	AHH_Mottakstank				: BOOL;
	HH_LS_Mottakstank			: BOOL;
	AHH_Reaktor					: BOOL;
	Reaktor_2_Forrigling		: BOOL;
END_VAR
VAR_OUTPUT
	PauseOK						: BOOL;
END_VAR
VAR

END_VAR


IF Pause THEN
	IF ((AHH_Mottakstank OR HH_LS_Mottakstank ) AND NOT Reaktor_2_Forrigling AND NOT AHH_Reaktor) THEN	// forrigling mot R2
		PauseOK := TRUE;
	ELSE
		PauseOK := FALSE;
	END_IF;
END_IF;

END_FUNCTION_BLOCK

// Device/Application/fbUtrekningar
FUNCTION_BLOCK fbUtrekningar
VAR_INPUT
END_VAR
VAR_OUTPUT
END_VAR
VAR
	Reaktor1		: MA;
	Reaktor2		: MA;
END_VAR



// Sette MA innganane

// Beregne frå nivå til volum reaktor 1
VolumReaktor(Height := GVL_R1.Nivaa, Volum => GVL_R1.Volum);

// Beregne frå nivå til volum reaktor 2
VolumReaktor(Height := GVL_R1.Nivaa, Volum => GVL_R2.Volum);

END_FUNCTION_BLOCK

// Device/Application/VolumReaktor
FUNCTION VolumReaktor : REAL
VAR_INPUT
	Height			: REAL;
END_VAR

VAR_OUTPUT
	Volum			: REAL;
END_VAR

VAR CONSTANT
	Radius 			: REAL := 3.0;
	pi_value 		: REAL := 3.14;
END_VAR


Volum := Height * pi_value * Radius * Radius;

END_FUNCTION

// Device/Application/Heile_R1/Reaktor1
PROGRAM Reaktor1
VAR

	Tilstandsmaskin		: tmReaktor;

	Innpumping			: R1_Innpumping;
	Pause				: R1_Pause;
	Reaksjon			: R1_Reaksjon;
	Sedementering		: R1_Sedementering;
	Uttaping			: R1_Uttapping;
	Beregning			: fbUtrekningar;
	Slam				: R1_Slam;
END_VAR

// Tilstander for Tilstandsmaskin
Pause(TM_Pause := Tilstandsmaskin.Pause); // R1_Pause
Innpumping(TM_Innpumping := Tilstandsmaskin.Innpumping); // R1_Innpumping
Reaksjon(TM_Reaksjon := Tilstandsmaskin.Reaksjon); // R1_Reaksjon
// Tilstandsmaskin for SARA Reaktor 1
Tilstandsmaskin(
    PauseOK := Pause.TM_PauseOK,
    InnpumpingOK := Innpumping.TM_InnpumpingOK,
    ReaksjonOK := Reaksjon.TM_ReaksjonOK,
    SedementeringOK := Sedementering.TM_SedementeringOK,
    UttappingOK := Uttaping.TM_UttappingOK); // tmReaktor
GVL_R1.Pause := Tilstandsmaskin.Pause;
GVL_R1.Innpumping := Tilstandsmaskin.Innpumping;
GVL_R1.Reaksjon := Tilstandsmaskin.Reaksjon;
GVL_R1.Sedimentering := Tilstandsmaskin.Sedementering;
GVL_R1.Uttapping := Tilstandsmaskin.Uttapping;
Sedementering(TM_Sedementering := Tilstandsmaskin.Sedementering); // R1_Sedementering
Uttaping(TM_Uttapping := Tilstandsmaskin.Uttapping); // R1_Uttapping
// Slamuttak
Slam(TM_Slam := Tilstandsmaskin.Reaksjon); // R1_Slam

END_PROGRAM

// Device/Application/Heile_R1/R1_Innpumping
FUNCTION_BLOCK R1_Innpumping
VAR_INPUT
	TM_Innpumping			: BOOL;
END_VAR
VAR_OUTPUT
	TM_InnpumpingOK			: BOOL;
END_VAR

VAR
PP00_LS02   		: MB;
PP00_LS01  			: MB;
PP00_LT01	 		: MA;
PP01_LT01	 		: MA;

PP01_PS01		 	: SBE;
PP02_PS01		 	: SBE;
PP01_VP01   		: SBV;

PA01_BL01				: SBE;

Sekvens_Innpumping	: fbInnpumping;
	Sim: FBVALVESIM;
END_VAR

VAR_TEMP
	PYHR			: REAL := 100;
	PYLR			: REAL := 0;
	PP00_LT01_PAHH	: REAL := 32;
	PP00_LT01_PALL	: REAL := 5;
	PP01_LT01_PAHH	: REAL := 90;
END_VAR

// -------------------------------------------------------------------------------------------------------------------------------- INPUTS --------------------------------------------------------------------------------------------------------------------------------
// Mottakstank vippe høg
PP00_LS01(); // MB
// Mottakstank vippe lav
PP00_LS02(); // MB
// Mottakstank Nivåmåling
PP00_LT01(
    X := GVL_Inputs.PP00_LT01_X,
    PAHH := PP00_LT01_PAHH,
    PALL := PP00_LT01_PALL,
    PYHR := PYHR,
    PYLR := PYLR); // MA
// Reaktor 1 Nivåmåling
PP01_LT01(X := GVL_Inputs.PP01_LT01_X, PAHH := PP01_LT01_PAHH, PYHR := PYHR, PYLR := PYLR); // MA
// -------------------------------------------------------------------------------------------------------------------------------- CODE --------------------------------------------------------------------------------------------------------------------------------
Sekvens_Innpumping(
    Sending_Tank_AHH := PP00_LT01.AHH,
    Sending_Tank_ALL := PP00_LT01.ALL,
    Sending_Tank_LS_High := PP00_LS01.Y,
    Sending_Tank_LS_Low := PP00_LS02.Y,
    Reciving_Tank_AHH := PP01_LT01.AHH,
    Reciving_Tank_ALL := PP01_LT01.ALL,
    ValveBCH := PP01_VP01.BCH,
    ValveBCL := PP01_VP01.BCL,
    Pump1BCL := PP01_PS01.BCL,
    Pump2BCL := PP02_PS01.BCL,
    TM_Innpumping := TM_Innpumping,
    Max_Innpumpings_Tid := GVL_R1.SekvenstidInnpumping,
    Intervall_blaser_tid := GVL_R1.IntervallBlaser,
    Gangtid_Blaser := GVL_R1.GangtidBlaser); // fbInnpumping
// Reaktor 1 blåser
PA01_BL01(
    XGH := PA01_BL01.Y,
    XH := Sekvens_Innpumping.Blower_start,
    XL := Sekvens_Innpumping.Blower_stopp,
    XE := Simu.XE,
    LA := Simu.LA); // SBE
GVL_Outputs.PA01_BL01_Y := PA01_BL01.Y;
TM_InnpumpingOK := Sekvens_Innpumping.TM_InnpumpingOK;
// -------------------------------------------------------------------------------------------------------------------------------- OUTPUTS --------------------------------------------------------------------------------------------------------------------------------
// Inntaktspumpe 1
PP01_PS01(
    XGH := PP01_PS01.Y,
    XH := Sekvens_Innpumping.Pump1XH,
    XL := Sekvens_Innpumping.Pump1XL,
    XE := Simu.XE,
    LA := Simu.LA); // SBE
GVL_Outputs.PP01_PS01_Y := PP01_PS01.Y;
// Inntaktspumpe 2
PP02_PS01(
    XGH := PP02_PS01.Y,
    XH := Sekvens_Innpumping.Pump2XH,
    XL := Sekvens_Innpumping.Pump2_XL,
    XE := Simu.XE,
    LA := Simu.LA); // SBE
GVL_Outputs.PP02_PS01_Y := PP02_PS01.Y;
// Reaktor 1 inn ventil
PP01_VP01(
    XGH := Sim.BCH,
    XGL := Sim.BCL,
    XH := Sekvens_Innpumping.Valve_Open,
    XL := Sekvens_Innpumping.Valve_Close,
    LA := Simu.LA); // SBV
Sim(X := PP01_VP01.Y); // FBVALVESIM

END_FUNCTION_BLOCK

// Device/Application/Heile_R1/R1_Pause
FUNCTION_BLOCK R1_Pause
VAR_INPUT
	XE					: BOOL;			// Input from state machine
END_VAR
VAR_OUTPUT
	Y					: BOOL;			// Output to state machine
END_VAR
VAR
	// INPUT BLOCKS
	PP00_LS02   		: MB;			// Mottasktank vippe lav, call "Monitor Binary" 
	PP00_LS01  			: MB;			// Mottasktank vippe høg, call "Monitor Binary" 
	PP00_LT01	 		: MA;			// Mottasktank nivåmålar, call "Monitor Analog"
	PP01_LT01	 		: MA;			// Reaktor 1 nivåmålar,   call "Monitor Analog"

	// OUTPUT BLOCKS
	PA01_BL01			: SBE;			// Reaktor 1 blåser,	 call "Switch Binary Electrical"
	
	// FUNCTION BLOCKS
	SekvensPause		: fbPause;		// Pause logic, call "fbPause"
END_VAR
VAR_TEMP
	// FUNCTION CONTROL PARAMETERS
	PYHR				: REAL := 100;	// (Mottasktank nivåmålar & Reaktor 1 nivåmålar) MA Parameter Y high range
	PYLR				: REAL := 0;	// (Mottasktank nivåmålar & Reaktor 1 nivåmålar) MA Parameter Y low range
	PP00_LT01_PAHH		: REAL := 70;	// (Mottasktank nivåmålar) 						 MA Parameter high high action
	PP01_LT01_PAHH		: REAL := 90;	// (Reaktor 1 nivåmålar)   						 MA Parameter low low action 
END_VAR

// -------------------------------------------------------------------------------------------------------------------------------------------------IN BLOCKS----------------------------------------------------------------------------------------------------------------------------------------------------------------------------------------------------------
// Mottakstank vippe høg
// INPUTS
PP00_LS01(X := GVL_Inputs.PP00_LS01_X); // MB
// Mottakstank vippe lav
// INPUTS
PP00_LS02(X := GVL_Inputs.PP00_LS02_X); // MB
// Mottakstank Nivåmåling
// INPUTS
PP00_LT01(X := GVL_Inputs.PP00_LT01_X, PAHH := PP00_LT01_PAHH, PYHR := PYHR, PYLR := PYLR); // MA
// OUTPUTS
// OUTPUTS
// OUTPUTS
GVL_Rest.MottakstankNivaa := PP00_LT01.Y;
// Reaktor 1 Nivåmåling
// INPUTS
PP01_LT01(X := GVL_Inputs.PP01_LT01_X, PAHH := PP01_LT01_PAHH, PYHR := PYHR, PYLR := PYLR); // MA
// OUTPUTS
GVL_R1.Nivaa := PP01_LT01.Y;
// -------------------------------------------------------------------------------------------------------------------------------------------------CODE ----------------------------------------------------------------------------------------------------------------------------------------------------------------------------------------------------------
SekvensPause(
    XE := XE,
    AHH_Mottakstank := PP00_LT01.AHH,
    AHH_LS_Mottakstank := PP00_LS01.Y,
    AHH_Reaktor := PP01_LT01.AHH,
    XB := GVL_R2.Innpumping,
    PTD := GVL_R1.GangtidBlaser,
    PTI := GVL_R1.IntervallBlaser); // fbPause
// -------------------------------------------------------------------------------------------------------------------------------------------------OUT BLOCKS----------------------------------------------------------------------------------------------------------------------------------------------------------------------------------------------------------
// Reaktor 1 Blåser
// Inputs
PA01_BL01(
    XGH := PA01_BL01.Y,
    XH := SekvensPause.YH_Blower,
    XL := SekvensPause.YL_Blower,
    XE := XE,
    LA := GVL_R1.Pause); // SBE
GVL_R1.Pause_PA01_BL01 := PA01_BL01.Y;
// OUTPUTS
GVL_R1.Pause_PA01_BL01_YF := PA01_BL01.YF;
Y := SekvensPause.Y;

END_FUNCTION_BLOCK

// Device/Application/Heile_R1/R1_Reaksjon
FUNCTION_BLOCK R1_Reaksjon
VAR_INPUT
	TM_Reaksjon			: BOOL;
END_VAR
VAR_OUTPUT
	TM_ReaksjonOK			: BOOL;
END_VAR
VAR
	Reaksjon				: fbReaksjon;
	Doseringspumpe			: SBE;
	Blaser					: SBE;
END_VAR

Reaksjon(
    TM_Reaksjon := TM_Reaksjon,
    Blaser_Confirmed_stopped := Blaser.BCL,
    Max_Reaksjon_Tid := GVL_R1.SekvenstidReaksjon,
    Gangtid_Anoks := GVL_R1.GangtidAnoks,
    Gangtid_Aerob := GVL_R1.GangtidAerob,
    Gangtid_Kjemikalie := GVL_R1.GangtidKjemikalieDosering,
    DoseringStartTidForSlutt := GVL_R1.SikkerheitsIntervallKjemikalie); // fbReaksjon
TM_ReaksjonOK := Reaksjon.TM_ReaksjonOK;
Blaser(XH := Reaksjon.Start_Blaser, XL := Reaksjon.Stopp_Blaser); // SBE
Doseringspumpe(XH := Reaksjon.Start_Pumpe, XL := Reaksjon.Stopp_Pumpe); // SBE

END_FUNCTION_BLOCK

// Device/Application/Function blocks/fbReaksjon
FUNCTION_BLOCK fbReaksjon
VAR_INPUT
	TM_Reaksjon							: BOOL;			// Start frå Tilstandsmaskin
	
	Blaser_Confirmed_stopped			: BOOL;
	
	// Timer og Tider
	Max_Reaksjon_Tid					: TIME;			// Sekvenstid
	Gangtid_Anoks						: TIME;			// Gangtid uten blåsing aktiv
	Gangtid_Aerob						: TIME;			// Gangtid med blåsing aktiv
	Gangtid_Kjemikalie					: TIME;			// Gangtid for kjemikalie
	DoseringStartTidForSlutt			: TIME;
END_VAR

VAR_OUTPUT
	TM_ReaksjonOK						: BOOL;			// Til Tilstandsmaskin
	
	// Blåser
	Start_Blaser						: BOOL;
	Stopp_Blaser						: BOOL;
	
	// Kjemikalie Pumpe
	Start_Pumpe							: BOOL;
	Stopp_Pumpe							: BOOL;
END_VAR

VAR
	AnoksTimer							: fbTimer;
	AerobTimer							: fbTimer;
	ReaksjonsTimer						: fbTimer;
	KjemikalieTimer						: fbTimer;
	
	siCase	: SINT;
END_VAR

VAR CONSTANT
	ciInit	: SINT := 0;
	ciAerob : SINT := 1;
	ciAnoks : SINT := 2;
END_VAR


// INPUTS

// Timer
AnoksTimer();
AerobTimer();
ReaksjonsTimer();
KjemikalieTimer();

AnoksTimer.PTDH 		:= Gangtid_Anoks;
AerobTimer.PTDH			:= Gangtid_Aerob;
ReaksjonsTimer.PTDH 	:= Max_Reaksjon_Tid;
KjemikalieTimer.PTDH	:= Max_Reaksjon_Tid - (Gangtid_Kjemikalie + DoseringStartTidForSlutt);
KjemikalieTimer.PTDL	:= Gangtid_Kjemikalie;

// Hantering av feil større ein max tid
IF (Gangtid_Anoks > Max_Reaksjon_Tid) THEN
	Gangtid_Anoks := Max_Reaksjon_Tid;
END_IF

IF (Gangtid_Aerob > Max_Reaksjon_Tid) THEN
	Gangtid_Aerob := Max_Reaksjon_Tid;
END_IF


IF TM_Reaksjon THEN
	
	CASE siCase OF
		
		ciInit:
		
		IF NOT (TM_ReaksjonOK) THEN
			ReaksjonsTimer.X 	:= TRUE;
			KjemikalieTimer.X 	:= TRUE;
			siCase := ciAerob;
		END_IF

		ciAerob:
			
			// Reset Anoks Timer
			AnoksTimer.X := FALSE;
			
			// Start Aerob Timer
			AerobTimer.X := TRUE;
			
			// Start Blåser
			Stopp_Blaser := FALSE;
			Start_Blaser := TRUE;
			
			// Neste case
			IF (AerobTimer.Y) THEN
				siCase := ciAnoks;
			END_IF
			
		ciAnoks:
		
			// Reset Aerob Timer
			AerobTimer.X := FALSE;
			
			// Start Anoks Timer
			AnoksTimer.X := TRUE;
			
			// Stopp Blåser
			Stopp_Blaser := TRUE;
			Start_Blaser := FALSE;
			
			// Neste case
			IF (AnoksTimer.Y) THEN
				siCase := ciAerob;
			END_IF
	END_CASE

	IF (KjemikalieTimer.Y) THEN
		
		KjemikalieTimer.X := FALSE;
		
		// Kjemikalie Pumpe
		Stopp_Pumpe := FALSE;
		Start_Pumpe := TRUE;

	ELSE
		// Kjemikalie Pumpe
		Stopp_Pumpe := TRUE;
		Start_Pumpe := FALSE;
	END_IF




	IF (ReaksjonsTimer.Y) THEN
		
		// Stopp blåser og pumpe uansett tilstand
		Stopp_Blaser := TRUE;
		Start_Blaser := FALSE;
					
		IF (Blaser_Confirmed_stopped) THEN
			
			// Reset Timers
			ReaksjonsTimer.X 	:= FALSE;
			KjemikalieTimer.X 	:= FALSE;
			AnoksTimer.X		:= FALSE;
			AerobTimer.X		:= FALSE;
			
			// Send to initial state
			siCase 				:= ciInit;
			
			// Send to tilstandsmaskin
			TM_ReaksjonOK 		:= TRUE;
		END_IF
	END_IF

ELSE
	TM_ReaksjonOK := FALSE;
END_IF


// OUTPUTS

END_FUNCTION_BLOCK

// Device/Application/Heile_R1/R1_Sedementering
FUNCTION_BLOCK R1_Sedementering
VAR_INPUT
	TM_Sedementering 	: BOOL; 			// Input from state machine
END_VAR
VAR_OUTPUT
	TM_SedementeringOK 	: BOOL;				// Output to state machine
END_VAR
VAR
	// INPUT BLOCKS

	// OUTPUT BLOCKS

	// FUNCTION BLOCKS	
	Sedimentering		: fbSedementering;	// Sedimentering logic, call "fbSedimentering"
END_VAR

// -------------------------------------------------------------------------------------------------------------------------------------------------IN BLOCKS----------------------------------------------------------------------------------------------------------------------------------------------------------------------------------------------------------
// ------------------------------------------------------------------------------------------------------------------------------------------------- CODE ----------------------------------------------------------------------------------------------------------------------------------------------------------------------------------------------------------
// ------------------------------------------------------------------------------------------------------------------------------------------------- OUT BLOCKS ----------------------------------------------------------------------------------------------------------------------------------------------------------------------------------------------------------
Sedimentering(TM_Sedementering := TM_Sedementering, SedementeringTid := GVL_R1.SekvenstidSedimentering); // fbSedementering
TM_SedementeringOK := Sedimentering.TM_SedementeringOK;

END_FUNCTION_BLOCK

// Device/Application/Function blocks/fbSedementering
FUNCTION_BLOCK fbSedementering
VAR_INPUT
	XE					: BOOL;		// External enable from state machine
END_VAR
VAR_INPUT RETAIN
	PST					: TIME;		// Parameter max sedimentation time
END_VAR

VAR_OUTPUT
	Y					: BOOL;		// Function output, pulsed true when sequence is finished.
END_VAR
VAR
	SedementeringTimer		: fbTimer;
END_VAR

// ***************************************************************************************
// Copyright: Peter Søreide Skaar, Roar Bøyum, Vegard Aven Ullebø [2024]
// All rights reserved.

// This code was developed as part of a Bachelor's thesis conducted for Renasys AS 
// and Sunnfjord Kommune. 

// Unauthorized reproduction, distribution, or modification of this code, in whole 
// or in part, is strictly prohibited without the express permission of the copyright 
// holder.
// ***************************************************************************************

SedementeringTimer();
SedementeringTimer.PTDH := PST;

IF (XE) THEN
	
	SedementeringTimer.X := TRUE;
	
	IF (SedementeringTimer.Y) THEN
		
		Y := TRUE;	
	END_IF
ELSE
	Y := FALSE;	
	SedementeringTimer.X := FALSE;
END_IF

END_FUNCTION_BLOCK

// Device/Application/Heile_R1/R1_Uttapping
FUNCTION_BLOCK R1_Uttapping
VAR_INPUT
	TM_Uttapping	: BOOL;
END_VAR
VAR_OUTPUT
	TM_UttappingOK	: BOOL;
END_VAR
VAR
	Uttapping		: fbUttapping;
	TW01_VP01		: SBV;
	PP01_LT01		: MA;
	Sim: FBVALVESIM;
END_VAR
VAR_TEMP
	PYHR			: REAL := 100;
	PYLR			: REAL := 0;
	PP00_LT01_PAHH	: REAL := 32;
	PP01_LT01_PAHH	: REAL := 90;
END_VAR

PP01_LT01(X := GVL_Inputs.PP01_LT01_X, PAHH := PP01_LT01_PAHH, PYHR := PYHR, PYLR := PYLR); // MA
Simu.R1Nivaa := PP01_LT01.Y;
Uttapping(
    TM_Uttapping := TM_Uttapping,
    Max_uttaping_Tid := GVL_R1.SekvenstidUttapping,
    Tank_ALL := PP01_LT01.ALL,
    Valve_Confirmed_Close := TW01_VP01.BCL,
    Reaktor_Nivaa := PP01_LT01.Y); // fbUttapping
TM_UttappingOK := Uttapping.TM_UttappingOK;
GVL_R1.DeltaNivaaDrenert := Uttapping.DeltaNivaa;
TW01_VP01(XGH := Sim.BCH, XGL := Sim.BCL, XH := Uttapping.Valve_Open, XL := Uttapping.Valve_Close); // SBV
Simu.TW02_VH01_YF := TW01_VP01.YF;
Sim(X := TW01_VP01.Y); // FBVALVESIM
GVL_Outputs.TW01_VP01_BCH := TW01_VP01.BCH;

END_FUNCTION_BLOCK

// Device/Application/Function blocks/fbUttapping
FUNCTION_BLOCK fbUttapping
VAR_INPUT
	X						: REAL;		// Input from leveltransmitter current level reactor
	XE						: BOOL;		// External enable from state machine
	XGL						: BOOL;		// Drain valve binary confirm low	
	X1						: BOOL;		// Low level from leveltransmitter reactor
END_VAR

VAR_INPUT RETAIN
	PUT						: TIME;		// Paramter Max uttapping time
END_VAR

VAR_OUTPUT
	Y						: BOOL;		// Output to state machine, pulsed if finshed sequence
	Y1						: REAL;		// Output (DeltaLevel) StartLevel - FinishedLevel
	YHDrainValve			: BOOL;		// Output YH open drain valve
	YLDrainValve			: BOOL;		// Output YL close drain valve
END_VAR
VAR
	UttappingTimer			: fbTimer;
	sbUttap					: BOOL;
	
	PreUttapNivaa			: REAL;
	sbFlank					: BOOL;
END_VAR

VAR_TEMP
	tbFlank					: BOOL;
END_VAR

// ***************************************************************************************
// Copyright: Peter Søreide Skaar, Roar Bøyum, Vegard Aven Ullebø [2024]
// All rights reserved.

// This code was developed as part of a Bachelor's thesis conducted for Renasys AS 
// and Sunnfjord Kommune. 

// Unauthorized reproduction, distribution, or modification of this code, in whole 
// or in part, is strictly prohibited without the express permission of the copyright 
// holder.
// ***************************************************************************************

// INNPUTS

// Timers
UttappingTimer();
UttappingTimer.PTDH := PUT;

IF (XE) THEN
	
	// Start av Timer
	UttappingTimer.X := TRUE;
	
	// Only posetiv edge
	IF (XE AND NOT sbUttap) THEN
		PreUttapNivaa := X;
	END_IF

	// Open valve
	YHDrainValve 	:= TRUE;
	YLDrainValve := FALSE;

	IF (X1 OR UttappingTimer.Y) THEN
		
		// Close valve
		YLDrainValve := TRUE;
		YHDrainValve  := FALSE;
		
		IF (XGL) THEN
			
			tbFlank := TRUE;
			
			// Reset Timer
			UttappingTimer.X := FALSE;
			
			// Til Tilstandsmaskin 
			Y := TRUE;
			
			IF (tbFlank AND NOT sbFLANK) THEN
				Y1 := PreUttapNivaa - X;
			END_IF
			
			// Posetive edge retrigger;
			sbFlank := tbFlank;
			
		END_IF		
	END_IF
ELSE
	tbFlank := FALSE;
	Y := FALSE;
END_IF

// Retrigger

sbUttap := XE;

// OUTPUTS

END_FUNCTION_BLOCK

// Device/Application/Heile_R1/R1_Slam
FUNCTION_BLOCK R1_Slam
VAR_INPUT
	TM_Slam : BOOL;	
END_VAR
VAR_OUTPUT
END_VAR
VAR
	fbslamutak	: fbSlamUtak;
	PS01_VP01 	: SBV;
	PS00_VP01 	: SBV; //Sivebedventil 1
	PS00_VP02 	: SBV; //Sivebedventil 2
	PS00_VP03 	: SBV; //Sivebedventil 3
	PS00_VP04 	: SBV; //Sivebedventil 4
	
	Sim1		: fbValveSim;
	Sim2		: fbValveSim;
	Sim3		: fbValveSim;
	Sim4		: fbValveSim;
	Sim5		: fbValveSim;
END_VAR

fbSlamutak(
    X1 := GVL_R1.Nivaa,
    X2 := GVL_Rest.siSivState,
    XE := TM_Slam,
    SivValve1BCL := PS00_VP01.BCL,
    SivValve2BCL := PS00_VP02.BCL,
    SivValve3BCL := PS00_VP03.BCL,
    SivValve4BCL := PS00_VP04.BCL,
    ReactorValveBCL := PS01_VP01.BCL,
    ReactorValveBCH := PS01_VP01.BCH,
    PTI := GVL_Rest.Uttaksintervall,
    PTMT := GVL_Rest.MaxGangtidSlam,
    PRAntattSlamNivaa := GVL_Rest.AntattSlamNivaa);
GVL_Rest.PulseCoutner := fbSlamutak.Y;
// -------------------------------------------------------------------------------------------------------------------------------- OUTPUTS --------------------------------------------------------------------------------------------------------------------------------
// Reaktor Slamventil
// INPUTS
PS01_VP01(XGH := Sim1.BCH, XGL := Sim1.BCL, XH := fbSlamutak.YHReactorValve, XL := fbSlamutak.YLReactorValve); // SBV
Sim1(X := PS01_VP01.Y); // fbValveSim
// OUTPUTS
GVL_Outputs.PS01_VP01_Y := PS01_VP01.Y;
GVL_R1.PS01_VP01_YF := PS01_VP01.YF;
// Sivebed1
// INPUTS
PS00_VP01(XGH := Sim2.BCH, XGL := Sim2.BCL, XH := fbSlamutak.YHSivbed1Valve, XL := fbSlamutak.YLSivbed1Valve); // SBV
Sim2(X := PS00_VP01.Y); // fbValveSim
// OUTPUTS
GVL_R1.PS00_VP01_Y := PS00_VP01.Y;
GVL_R1.PS00_VP01_YF := PS00_VP01.YF;
// Sivebed2
// INPUTS
PS00_VP02(XGH := Sim3.BCH, XGL := Sim3.BCL, XH := fbSlamutak.YHSivbed2Valve, XL := fbSlamutak.YLSivbed2Valve); // SBV
Sim3(X := PS00_VP02.Y); // fbValveSim
// OUTPUTS
GVL_R1.PS00_VP02_Y := PS00_VP02.Y;
GVL_R1.PS00_VP02_YF := PS00_VP02.YF;
// Sivebed3
// INPUTS
PS00_VP03(XGH := Sim4.BCH, XGL := Sim4.BCL, XH := fbSlamutak.YHSivbed3Valve, XL := fbSlamutak.YLSivbed3Valve); // SBV
Sim4(X := PS00_VP03.Y); // fbValveSim
// OUTPUTS
GVL_R1.PS00_VP03_Y := PS00_VP03.Y;
GVL_R1.PS00_VP03_YF := PS00_VP03.YF;
// Sivebed4
// INPUTS
PS00_VP04(XGH := Sim4.BCH, XGL := Sim4.BCL, XH := fbSlamutak.YHSivbed4Valve, XL := fbSlamutak.YLSivbed4Valve); // SBV
Sim4(X := PS00_VP04.Y); // fbValveSim
// OUTPUTS
GVL_R1.PS00_VP04_Y := PS00_VP04.Y;
GVL_R1.PS00_VP04_YF := PS00_VP04.YF;

END_FUNCTION_BLOCK

// Device/Application/Function blocks/fbSlamutak
FUNCTION_BLOCK fbSlamutak
VAR_INPUT
	TM_Slamutak					: BOOL;	
	
	Slamalder					: INT;
	AntattSlamNivaa				: REAL;
			
	ReactorLevel				: REAL;

	SivValve1BCL				: BOOL;
	SivValve2BCL				: BOOL;
	SivValve3BCL				: BOOL;
	SivValve4BCL				: BOOL;
	
	ReactorValveBCL				: BOOL;
	ReactorValveBCH				: BOOL;
	
	Uttaksintervall				: TIME;
	MaxGangTidSlamUtak			: TIME;	
END_VAR

VAR_OUTPUT
	Y							: BOOL; //Sender pulse ferdig til sivbedHandtering for telling
	Open_Reactor_Valve			: BOOL;
	Close_Reactor_Valve			: BOOL;
	
	Open_SivCelle_1_Valve		: BOOL;
	Close_SivCelle_1_Valve		: BOOL;
	
 	Open_SivCelle_2_Valve		: BOOL;
 	Close_SivCelle_2_Valve		: BOOL;
 	
 	Open_SivCelle_3_Valve		: BOOL;
 	Close_SivCelle_3_Valve		: BOOL;
 	
 	Open_SivCelle_4_Valve		: BOOL;
 	Close_SivCelle_4_Valve		: BOOL;

END_VAR

VAR
	siSivBed					: SINT;	
	PreUttakNiva				: REAL;	
	sbUttakTimerY				: BOOL;	
	
	GangtidSlamtapping			: fbTimer;
	UttaksTimer					: fbTimer;
	SivBedTimer					: fbTimer;
	OutputPulse					: fbTimer;

	CmSlamUttak					: REAL;
	
	AktivSivCelleBCL			: BOOL;
	
END_VAR

VAR_TEMP
	tiMillis						: LINT;
	tiDays							: LINT;
END_VAR

VAR CONSTANT
	ciInit			: SINT := 0;
	ciCelle1		: SINT := 1;
	ciCelle2		: SINT := 2;
	ciCelle3		: SINT := 3;
	CiCelle4		: SINT := 4;
	PTD				: TIME := T#2S;
	
	cliMillis2Days	: LINT := 86400000;	
	
END_VAR


// Timer teller kontinuerlig om
UttaksTimer();
GangtidSlamTapping();
OutputPulse();


UttaksTimer.PTDH := Uttaksintervall;
GangtidSlamTapping.PTDH := MaxGangTidSlamUtak;
OutputPulse.PTDL := PTD;
UttaksTimer.X := TRUE;
OutputPulse.X := FALSE;

// Convert TIME to days in INT.
tiMillis := TIME_TO_INT(Uttaksintervall);
tiDays := tiMillis / cliMillis2Days;

IF (TM_Slamutak) THEN
	
	// Timer goes true and begins slamuttak
	IF (UttaksTimer.Y) THEN
		
		// Storing level of reactor tank before opening valves on posetive edge		
		IF (UttaksTimer.Y AND NOT sbUttakTimerY) THEN			
			cmSlamUttak := (tiDays * AntattSlamNivaa)/Slamalder; 	// Calculating slamuttak			
			PreUttakNiva := ReactorLevel;							// Store Reactorlevel before started sludge removal.
			GangtidSlamtapping.X := TRUE;							// Start timer 			
		END_IF		
		
		// Opne reaktor slam ventil		
		Open_Reactor_Valve := TRUE;
		Close_Reactor_Valve := FALSE;
		
		// Based on which sivcelle is in use open the respectiv valves
		// Required Reactorvalve confirmed open		
		IF (ReactorValveBCH) THEN
		
			IF (siSivBed = ciCelle1) THEN
			
				Close_Sivcelle_1_Valve 		:= FALSE;
				Open_Sivcelle_1_Valve 		:= TRUE;
			
			ELSIF (siSivBed = ciCelle2) THEN
			
				Close_Sivcelle_2_Valve 		:= FALSE;
				Open_Sivcelle_2_Valve 		:= TRUE;
			
			ELSIF (siSivBed = ciCelle3) THEN
			
				Close_Sivcelle_3_Valve 		:= FALSE;
				Open_Sivcelle_3_Valve 		:= TRUE;
		
			ELSIF (siSivBed = ciCelle4) THEN
				
				Close_Sivcelle_4_Valve 		:= FALSE;
				Open_Sivcelle_4_Valve 		:= TRUE;
			END_IF		
		END_IF
		
		// Stopping SlamUttak when the required amout of sludge is removed from the reactor
		
		IF ((ReactorLevel < (PreUttakNiva - CmSlamUttak)) OR GangTidSlamTapping.Y) THEN
			
			// Closing reactor valve
			
			Open_Reactor_Valve 		:= FALSE;
			Close_Reactor_Valve 	:= TRUE;
						
			// Closing sivcelle valves 			
			IF    (siSivBed = ciCelle1) THEN
			
				AktivSivCelleBCL := SivValve1BCL;
			
				Close_Sivcelle_1_Valve 		:= TRUE;
				Open_Sivcelle_1_Valve 		:= FALSE;
			
			ELSIF (siSivBed = ciCelle2) THEN
			
				AktivSivCelleBCL := SivValve2BCL;
			
				Close_Sivcelle_2_Valve 		:= TRUE;
				Open_Sivcelle_2_Valve 		:= FALSE;
			
			ELSIF (siSivBed = ciCelle3) THEN
			
				AktivSivCelleBCL := SivValve3BCL;
			
				Close_Sivcelle_3_Valve 		:= TRUE;
				Open_Sivcelle_3_Valve 		:= FALSE;
		
			ELSIF (siSivBed = ciCelle4) THEN
				
				AktivSivCelleBCL := SivValve4BCL;
				
				Close_Sivcelle_4_Valve 		:= TRUE;
				Open_Sivcelle_4_Valve 		:= FALSE;
			END_IF
				
				
			// If the vales are confirmed close the initial timer is reset and starts counting again		
			IF ((ReactorValveBCL AND AktivSivCelleBCL)) THEN
			
			// Resetting timer
			UttaksTimer.X 			:= FALSE;
			GangtidSlamtapping.X 	:= FALSE;			
			OutputPulse.X := TRUE;					
			END_IF		
		END_IF		
	END_IF
	
	// Posetive edge retrigger
	sbUttakTimerY := UttaksTimer.Y;	
END_IF



//Handle outputs
Y := OutputPulse.Y;

END_FUNCTION_BLOCK

// Device/Application/Heile_R2/Reaktor2
PROGRAM Reaktor2
VAR
	Tilstandsmaskin		: tmReaktor;
	Innpumping			: R1_Innpumping;
	Pause				: R1_Pause;
	Reaksjon			: R1_Reaksjon;
	Sedementering		: R1_Sedementering;
	Uttaping			: R1_Uttapping;
	Beregning			: fbCalculations;	
END_VAR

// Tilstander for Tilstandsmaskin
Pause(XE := Tilstandsmaskin.Pause); // R1_Pause
Innpumping(XE := Tilstandsmaskin.Innpumping); // R1_Innpumping
Reaksjon(XE := Tilstandsmaskin.Reaksjon); // R1_Reaksjon
// Tilstandsmaskin for SARA Reaktor 1
Tilstandsmaskin(
    PauseOK := Pause.Y,
    InnpumpingOK := Innpumping.Y,
    ReaksjonOK := Reaksjon.Y,
    SedementeringOK := Sedementering.Y,
    UttappingOK := Uttaping.Y); // tmReaktor
GVL_R1.Pause := Tilstandsmaskin.Pause;
GVL_R1.Innpumping := Tilstandsmaskin.Innpumping;
GVL_R1.Reaksjon := Tilstandsmaskin.Reaksjon;
GVL_R1.Sedimentering := Tilstandsmaskin.Sedementering;
GVL_R1.Uttapping := Tilstandsmaskin.Uttapping;
GVL_R1.State := Tilstandsmaskin.State;
Sedementering(XE := Tilstandsmaskin.Sedementering); // R1_Sedementering
Uttaping(XE := Tilstandsmaskin.Uttapping); // R1_Uttapping

END_PROGRAM

// Device/Application/Heile_R2/Reaktor2
PROGRAM Reaktor2
VAR
	Tilstandsmaskin		: tmReaktor;

	Innpumping			: R2_Innpumping;
	Pause				: R2_Pause;
END_VAR

Tilstandsmaskin(PauseOK := Pause.TM_PauseOK, InnpumpingOK := Innpumping.TM_InnpumpingOK); // tmReaktor
GVL_TM.R2_Pause := Tilstandsmaskin.Pause;
GVL_TM.R2_Innpumping := Tilstandsmaskin.Innpumping;
GVL_TM.R2_Reaksjon := Tilstandsmaskin.Reaksjon;
GVL_TM.R2_Sedementering := Tilstandsmaskin.Sedementering;
GVL_TM.R2_Uttapping := Tilstandsmaskin.Uttapping;
Innpumping(TM_Innpumping := Tilstandsmaskin.Innpumping); // R2_Innpumping
Pause(TM_Pause := Tilstandsmaskin.Pause); // R2_Pause

END_PROGRAM

// Device/Application/Heile_R2/R2_Pause
FUNCTION_BLOCK R2_Pause
VAR_INPUT
	XE					: BOOL;			// Input from state machine
END_VAR
VAR_OUTPUT
	Y					: BOOL;			// Output to state machine
END_VAR
VAR
	// INPUT BLOCKS
	PP00_LS02   		: MB;			// Mottasktank vippe lav, call "Monitor Binary" 
	PP00_LS01  			: MB;			// Mottasktank vippe høg, call "Monitor Binary" 
	PP00_LT01	 		: MA;			// Mottasktank nivåmålar, call "Monitor Analog"
	PP02_LT02	 		: MA;			// Reaktor 2 nivåmålar,   call "Monitor Analog"

	// OUTPUT BLOCKS
	PA02_BL01			: SBE;			// Reaktor 2 blåser,	 call "Switch Binary Electrical"
	
	// FUNCTION BLOCKS
	SekvensPause		: fbPause;		// Pause logic, call "fbPause"	
	PA02_BL0			: SBE;
END_VAR
VAR_TEMP
	// FUNCTION CONTROL PARAMETERS
	PYHR				: REAL := 100;	// (Mottasktank nivåmålar & Reaktor 1 nivåmålar) MA Parameter Y high range
	PYLR				: REAL := 0;	// (Mottasktank nivåmålar & Reaktor 1 nivåmålar) MA Parameter Y low range
	PP00_LT01_PAHH		: REAL := 32;	// (Mottasktank nivåmålar) 						 MA Parameter high high action
	PP02_LT02_PAHH		: REAL := 90;	// (Reaktor 2 nivåmålar)   						 MA Parameter low low action 
END_VAR

// -------------------------------------------------------------------------------------------------------------------------------------------------IN BLOCKS----------------------------------------------------------------------------------------------------------------------------------------------------------------------------------------------------------
// Mottakstank vippe høg
// INPUTS
PP00_LS01(X := GVL_Inputs.PP00_LS01_X); // MB
// Mottakstank vippe lav
// INPUTS
PP00_LS02(X := GVL_Inputs.PP00_LS02_X); // MB
// Mottakstank Nivåmåling
// INPUTS
PP00_LT01(X := GVL_Inputs.PP00_LT01_X, PAHH := PP00_LT01_PAHH, PYHR := PYHR, PYLR := PYLR); // MA
// OUTPUTS
// OUTPUTS
// OUTPUTS
GVL_Rest.MottakstankNivaa := PP00_LT01.Y;
// Reaktor 2 Nivåmåling
// INPUTS
PP02_LT02(X := GVL_Inputs.PP02_LT02_X, PAHH := PP02_LT02_PAHH, PYHR := PYHR, PYLR := PYLR); // MA
// OUTPUTS
GVL_R2.Nivaa := PP02_LT02.Y;
// -------------------------------------------------------------------------------------------------------------------------------------------------CODE ----------------------------------------------------------------------------------------------------------------------------------------------------------------------------------------------------------
SekvensPause(
    XE := XE,
    AHH_Mottakstank := PP00_LT01.AHH,
    AHH_LS_Mottakstank := PP00_LS01.Y,
    AHH_Reaktor := PP02_LT02.AHH,
    XB := GVL_R1.Innpumping,
    PTD := GVL_R2.GangtidBlaser,
    PTI := GVL_R2.IntervallBlaser); // fbPause
// -------------------------------------------------------------------------------------------------------------------------------------------------OUT BLOCKS----------------------------------------------------------------------------------------------------------------------------------------------------------------------------------------------------------
// Reaktor 2 Blåser
// Inputs
PA02_BL01(
    XGH := PA02_BL01.Y,
    XH := SekvensPause.YH_Blower,
    XL := SekvensPause.YL_Blower,
    XE := XE,
    LA := GVL_R2.Pause); // SBE
GVL_R2.Pause_PA01_BL01 := PA02_BL01.Y;
// OUTPUTS
GVL_R2.Pause_PA01_BL01_YF := PA02_BL01.YF;
Y := SekvensPause.Y;

END_FUNCTION_BLOCK

// Device/Application/Heile_R2/R2_Pause
FUNCTION_BLOCK R2_Pause
VAR_INPUT
	TM_Pause			: BOOL;
END_VAR
VAR_OUTPUT
	TM_PauseOK			: BOOL;
END_VAR
VAR
	PP00_LS01	: MB;
	PP00_LS02	: MB;
	PP00_LT01	: MA;
	PP01_LT01	: MA;
	
	SekvensPause	: fbPause;	
END_VAR

PP00_LS01(); // MB
PP00_LS02(); // MB
PP00_LT01(); // MA
PP01_LT01(); // MA
SekvensPause(
    Pause := TM_Pause,
    AHH_Mottakstank := PP00_LT01.AHH,
    HH_LS_Mottakstank := PP00_LS01.Y,
    AHH_Reaktor := PP01_LT01.AHH,
    Reaktor_2_Forrigling := GVL_TM.R1_Innpumping); // fbPause
TM_PauseOK := SekvensPause.PauseOK;

END_FUNCTION_BLOCK

// Device/Application/Heile_R2/R2_Innpumping
FUNCTION_BLOCK R2_Innpumping
VAR_INPUT
	TM_Innpumping			: BOOL;
END_VAR
VAR_OUTPUT
	TM_InnpumpingOK			: BOOL;
END_VAR

VAR
PP00_LS02   		: MB;
PP00_LS01  			: MB;
PP00_LT01	 		: MA;
PP01_LT01	 		: MA;

PP01_PS01		 	: SBE;
PP02_PS01		 	: SBE;
PP01_VP01   		: SBV;

Sekvens_Innpumping	: fbInnpumping;

END_VAR

PP00_LS01(); // MB
PP00_LS02(); // MB
PP00_LT01(); // MA
PP01_LT01(); // MA
Sekvens_Innpumping(
    Sending_Tank_AHH := PP00_LT01.AHH,
    Sending_Tank_ALL := PP00_LT01.ALL,
    Sending_Tank_LS_High := PP00_LS01.Y,
    Sending_Tank_LS_Low := PP00_LS02.Y,
    Reciving_Tank_AHH := PP01_LT01.AHH,
    Reciving_Tank_ALL := PP01_LT01.ALL,
    ValveBCH := PP01_VP01.BCH,
    ValveBCL := PP01_VP01.BCL,
    Pump1BCL := PP01_PS01.BCL,
    Pump2BCL := PP02_PS01.BCL,
    TM_Innpumping := TM_Innpumping); // fbInnpumping
TM_InnpumpingOK := Sekvens_Innpumping.TM_InnpumpingOK;
PP01_VP01(XH := Sekvens_Innpumping.Valve_Open, XL := Sekvens_Innpumping.Valve_Close); // SBV
PP01_PS01(XH := Sekvens_Innpumping.Pump1XH, XL := Sekvens_Innpumping.Pump1XL); // SBE
PP02_PS01(XH := Sekvens_Innpumping.Pump2XH, XL := Sekvens_Innpumping.Pump2_XL); // SBE

END_FUNCTION_BLOCK

// Device/Application/Heile_R2/R2_Innpumping
FUNCTION_BLOCK R2_Innpumping
VAR_INPUT
	XE						: BOOL;			// Input from state machine
END_VAR
VAR_OUTPUT
	Y						: BOOL;			// Output to state machine
END_VAR

VAR
	// INPUT BLOCKS
	PP00_LS02   			: MB;			// Mottasktank vippe lav, call "Monitor Binary" 
	PP00_LS01  				: MB;			// Mottasktank vippe høg, call "Monitor Binary" 
	PP00_LT01	 			: MA;			// Mottasktank nivåmålar, call "Monitor Analog"
	PP01_LT01	 			: MA;			// Reaktor 2 nivåmålar,   call "Monitor Analog"
	
	// OUTPUT BLOCKS
	PA01_BL01				: SBE;			// Reaktor 2 blåser,	 call "Switch Binary Electrical"
	PP01_PS01		 		: SBE;			// Matepumpe 1,			 call "Switch Binary Electrical"
	PP02_PS01		 		: SBE;			// Matepumpe 2,			 call "Switch Binary Electrical"
	PP01_VP01   			: SBV;			// Reaktor 2 inn ventil, call "Switch Binary Valve"
	
	// FUNCTION BLOCKS
	Sekvens_Innpumping		: fbInnpumping;	// Innpumping logic,         call "fbInnpumping"
	Sim						: fbValveSim;	// Feedback balve simulator, call "fbValveSim"
	PA02_BL01				: SBE;
	PP02_VP01				: SBV;
	PP02_LT02				: MA;

END_VAR

VAR_TEMP		
	// FUNCTION CONTROL PARAMETERS
	PYHR					: REAL := 100;		// (Mottasktank nivåmålar & Reaktor 2 nivåmålar) MA Parameter Y high range
	PYLR					: REAL := 0;		// (Mottasktank nivåmålar & Reaktor 2 nivåmålar) MA Parameter Y low range
	PP00_LT01_PBXH			: REAL := 70;		// (Mottasktank nivåmålar) 						 MA Parameter high high action
	PP00_LT01_PBXL			: REAL := 10;		// (Mottasktank nivåmålar) 						 MA Parameter low low action
	PP02_LT02_PBXH			: REAL := 90;		// (Reaktor 2 nivåmålar)   						 MA Parameter high high action
	END_VAR

// -------------------------------------------------------------------------------------------------------------------------------------------------IN BLOCKS----------------------------------------------------------------------------------------------------------------------------------------------------------------------------------------------------------
// Mottakstank vippe høg
// INPUTS
// OUTPUTS
PP00_LS01(X := GVL_Inputs.PP00_LS01_X); // MB
// Mottakstank vippe lav
// INPUTS
PP00_LS02(X := GVL_Inputs.PP00_LS02_X); // MB
// Mottakstank Nivåmåling
// INPUTS
PP00_LT01(
    X := GVL_Inputs.PP00_LT01_X,
    PBXH := PP00_LT01_PBXH,
    PBXL := PP00_LT01_PBXL,
    PYHR := PYHR,
    PYLR := PYLR); // MA
// OUTPUTS
// OUTPUTS
GVL_Rest.MottakstankNivaa := PP00_LT01.Y;
// Reaktor 2 Nivåmåling
// INPUTS
PP02_LT02(X := GVL_Inputs.PP02_LT02_X, PBXH := PP02_LT02_PBXH, PYHR := PYHR, PYLR := PYLR); // MA
// OUTPUTS
GVL_R2.Nivaa := PP02_LT02.Y;
// ------------------------------------------------------------------------------------------------------------------------------------------------- CODE ----------------------------------------------------------------------------------------------------------------------------------------------------------------------------------------------------------
Sekvens_Innpumping(
    X1_SendingTank := PP00_LT01.BXH,
    X2_SendingTank := PP00_LT01.BXL,
    X3_SendingTank := PP00_LS01.Y,
    X4_Sending_Tank := PP00_LS02.Y,
    X5_ReceivingTank := PP02_LT02.BXH,
    X6_ReceivingTank := PP02_LT02.BXL,
    X7_RValve := PP02_VP01.BCH,
    X8_RValve := PP02_VP01.BCL,
    X9_Pump1 := PP01_PS01.BCL,
    X10_Pump2 := PP02_PS01.BCL,
    XE := XE,
    PIT := GVL_R2.SekvenstidInnpumping,
    PTI := GVL_R2.IntervallBlaser,
    PTD := GVL_R2.GangtidBlaser); // fbInnpumping
// Reaktor 2 blåser
// INPUTS
PA02_BL01(
    XGH := PA02_BL01.Y,
    XH := Sekvens_Innpumping.YH_Blower,
    XL := Sekvens_Innpumping.YL_Blower,
    XE := GVL_R2.Innpumping,
    LA := Simu.LA); // SBE
GVL_R2.Innpumping_PA01_BL01_YF := PA02_BL01.YF;
Y := Sekvens_Innpumping.Y;
// ------------------------------------------------------------------------------------------------------------------------------------------------- OUT BLOCKS  ----------------------------------------------------------------------------------------------------------------------------------------------------------------------------------------------------------
// Inntaktspumpe 1
// INPUTS
PP01_PS01(
    XGH := PP01_PS01.Y,
    XH := Sekvens_Innpumping.YH_Pump1,
    XL := Sekvens_Innpumping.YL_Pump1,
    XE := GVL_R2.Innpumping,
    LA := Simu.LA); // SBE
GVL_R2.PP01_PS01_YF := PP01_PS01.YF;
// OUTPUTS
GVL_R2.PP01_PS01_Y := PP01_PS01.Y;
// Inntaktspumpe 2
// INPUTS
PP02_PS01(
    XGH := PP02_PS01.Y,
    XH := Sekvens_Innpumping.YH_Pump2,
    XL := Sekvens_Innpumping.YL_Pump2,
    XE := GVL_R2.Innpumping,
    LA := Simu.LA); // SBE
// OUTPUTS
GVL_R2.PP02_PS01_Y := PP02_PS01.Y;
GVL_R2.PP02_PS01_YF := PP02_PS01.YF;
// OUTPUTS
GVL_R2.Innpumping_PA02_BL01 := PA02_BL01.Y;
// Reaktor 2 inn ventil
// INPUTS
PP02_VP01(
    XGH := Sim.BCH,
    XGL := Sim.BCL,
    XH := Sekvens_Innpumping.YH_RValve,
    XL := Sekvens_Innpumping.YL_RValve,
    LA := Simu.LA); // SBV
// OUTPUTS
GVL_Outputs.PP02_VP01_Y := PP02_VP01.Y;
GVL_R2.PP01_VP01_YF := PP02_VP01.YF;
GVL_R2.PP01_VP01_BCH := PP02_VP01.BCH;
Sim(X := PP02_VP01.Y); // FBVALVESIM

END_FUNCTION_BLOCK

// Device/Application/Heile_R2/R2_Reaksjon
FUNCTION_BLOCK R2_Reaksjon
VAR_INPUT
	XE					: BOOL;			// Input from state machine
END_VAR
VAR_OUTPUT
	Y					: BOOL; 		// Output to state machine
END_VAR
VAR
	// INPUT BLOCKS

	// OUTPUT BLOCKS
	CH00_PH01			: SBE;			// Reaktor 2 doseringspumpe, call "Switch Binary Electrical"
	PA01_BL01			: SBE;			// Reaktor 2 blåser,	 	 call "Switch Binary Electrical"
	Slam				: R1_Slam;		// Slammuttak
	
	// FUNCTION BLOCKS
	Reaksjon			: fbReaksjon;	// Reaksjon logic, call "fbReaksjon"
	PA02_BL01			: SBE;			// Blower R2
	CH00_PH02			: SBE;			// ChemPump R2
END_VAR

// note: 2 stored wires end on pins the file does not list and are not shown
// Slamuttak
Slam(XE := XE); // R1_Slam
// -------------------------------------------------------------------------------------------------------------------------------------------------IN BLOCKS----------------------------------------------------------------------------------------------------------------------------------------------------------------------------------------------------------
// ------------------------------------------------------------------------------------------------------------------------------------------------- CODE ----------------------------------------------------------------------------------------------------------------------------------------------------------------------------------------------------------
Reaksjon(
    XE := XE,
    XHLBlower := PA02_BL01.BCL,
    PRT := GVL_R2.SekvenstidReaksjon,
    PTAN := GVL_R2.GangtidAnoks,
    PTAE := GVL_R2.GangtidAerob,
    PTCP := GVL_R2.GangtidKjemikalieDosering,
    PTCR := GVL_R2.SikkerheitsIntervallKjemikalie); // fbReaksjon
Y := Reaksjon.Y;
// ------------------------------------------------------------------------------------------------------------------------------------------------- OUT BLOCKS ----------------------------------------------------------------------------------------------------------------------------------------------------------------------------------------------------------
// Reaktor 2 Blåser
// INPUTS
PA02_BL01(XH := Reaksjon.YHBlower, XL := Reaksjon.YLBlower, XE := GVL_R2.Reaksjon, LA := Simu.LA); // SBE
GVL_R2.Reaksjon_PA01_BL01_YF := PA02_BL01.YF;
// OUTPUTS
GVL_R2.Reaksjon_PA01_BL01 := PA02_BL01.Y;
// Reaktor 2 Doseringspumpe
// INPUTS
CH00_PH02(
    XGH := CH00_PH02.Y,
    XH := Reaksjon.YHChemPump,
    XL := Reaksjon.YLChemPump,
    XE := GVL_R2.Reaksjon,
    LA := Simu.LA); // SBE
GVL_R2.CH00_PH02_YF := CH00_PH02.YF;
// OUTPUTS
GVL_Outputs.CH00_PH02_Y := CH00_PH02.Y;

END_FUNCTION_BLOCK

// Device/Application/Heile_R2/R2_Sedementering
FUNCTION_BLOCK R2_Sedementering
VAR_INPUT
	XE 					: BOOL; 			// Input from state machine
END_VAR
VAR_OUTPUT
	Y 					: BOOL;				// Output to state machine
END_VAR
VAR
	// INPUT BLOCKS

	// OUTPUT BLOCKS

	// FUNCTION BLOCKS	
	Sedimentering		: fbSedementering;	// Sedimentering logic, call "fbSedimentering"
END_VAR

// -------------------------------------------------------------------------------------------------------------------------------------------------IN BLOCKS----------------------------------------------------------------------------------------------------------------------------------------------------------------------------------------------------------
// ------------------------------------------------------------------------------------------------------------------------------------------------- CODE ----------------------------------------------------------------------------------------------------------------------------------------------------------------------------------------------------------
// ------------------------------------------------------------------------------------------------------------------------------------------------- OUT BLOCKS ----------------------------------------------------------------------------------------------------------------------------------------------------------------------------------------------------------
Sedimentering(XE := XE, PST := GVL_R2.SekvenstidSedimentering); // fbSedementering
Y := Sedimentering.Y;

END_FUNCTION_BLOCK

// Device/Application/Heile_R2/R2_Uttapping
FUNCTION_BLOCK R2_Uttapping
VAR_INPUT
	XE	: BOOL;				 // Input from state machine
END_VAR
VAR_OUTPUT
	Y				: BOOL; // Output to state machine
END_VAR
VAR
	// INPUT BLOCKS
	PP01_LT01		: MA; 	// Reaktor 1 nivåmålar,   call "Monitor Analog"
	
	// OUTPUT BLOCKS
	TW01_VP01		: SBV;	// Reaktor 1 dreneringsventil, call "Switch Binary Valve"
	
	// FUNCTION BLOCKS
	Uttapping		: fbUttapping;
	Sim				: FBVALVESIM;
	PP02_LT02		: MA;
	TW02_VP01		: SBV;
	PP02_LT022_PALL: INT;
END_VAR
VAR_TEMP
	PYHR			: REAL := 100;
	PYLR			: REAL := 0;	
	PP02_LT02_PAHH	: REAL := 90;
	PP02_LT02_PALL	: REAL := 90;
	
END_VAR

// ------------------------------------------------------------------------------------------------------------------------------------------------- IN BLOCKS ----------------------------------------------------------------------------------------------------------------------------------------------------------------------------------------------------------
// Reaktor 2 Nivåmålar
// INPUTS
PP02_LT02(
    X := GVL_Inputs.PP02_LT02_X,
    PAHH := PP02_LT02_PAHH,
    PALL := PP02_LT022_PALL,
    PYHR := PYHR,
    PYLR := PYLR); // MA
// OUTPUTS
GVL_R2.Nivaa := PP02_LT02.Y;
// ------------------------------------------------------------------------------------------------------------------------------------------------- CODE  ----------------------------------------------------------------------------------------------------------------------------------------------------------------------------------------------------------
Uttapping(
    XE := XE,
    PUT := GVL_R2.SekvenstidUttapping,
    ALL := PP02_LT02.ALL,
    XGL := TW02_VP01.BCL,
    X := PP02_LT02.Y); // fbUttapping
Y := Uttapping.Y;
GVL_R2.DeltaNivaaDrenert := Uttapping.Y1;
// ------------------------------------------------------------------------------------------------------------------------------------------------- OUTPUT BLOCKS ----------------------------------------------------------------------------------------------------------------------------------------------------------------------------------------------------------
// Reaktor 2 dreneringsventil
// INPUTS
TW02_VP01(
    XGH := Sim.BCH,
    XGL := Sim.BCL,
    XH := Uttapping.YHDrainValve,
    XL := Uttapping.YLDrainValve,
    LA := Simu.LA); // SBV
GVL_R2.TW01_VH01_YF := TW02_VP01.YF;
Sim(X := TW02_VP01.Y); // FBVALVESIM
// OUTPUTS
GVL_Outputs.TW02_VP01_Y := TW02_VP01.Y;

END_FUNCTION_BLOCK

// Device/Application/IEC_Time
FUNCTION IEC_Time : BOOL
VAR_INPUT
	Start : BOOL;
END_VAR

VAR
END_VAR

END_FUNCTION

// Device/Application/POU
PROGRAM POU
VAR
	test : BOOL;
	test2 : BOOL;
END_VAR

END_PROGRAM

// Device/Application/SBV_ReArranged
FUNCTION_BLOCK SBV_ReArranged
VAR_INPUT
	XGH            : BOOL;                		 // eXternal Feedback Position High
    XGL            : BOOL;                		 // eXternal Feedback Position Low
    XH             : BOOL;                		 // eXternal Switch to Position High - in automatic mode
    XL             : BOOL;                		 // eXternal Switch to Position Low - in automatic mode
	XOH            : BOOL;               		 // eXternal Switch to Posistion High - in local/outside mode
	XOL            : BOOL;               		 // eXternal Switch to Posistion Low - in local/outside mode
	XF             : BOOL;                 		 // eXternal Fault 
	LSH            : BOOL;               		 // Lock Safeguard High
	LSL            : BOOL;               		 // Lock Safeguard Low
	FSH            : BOOL;                		 // Force Safeguarding High
    FSL            : BOOL;                		 // [Priority] Force Safeguarding Low
    FDH            : BOOL;              		 // Force Disable High
    FDL            : BOOL;             		     // [Priority] Force Disable Low
	FB             : BOOL;             		     // Force Block	
	FU             : BOOL;						 // Force Supression
	LA             : BOOL;               		 // Set Auto
	LM             : BOOL;               		 // [Priority 2]Set Manual
	LO             : BOOL;               		 // [Priority 1]Set Outside
    //RX             : BOOL;               		 // Reset Fault	
END_VAR

VAR_INPUT RETAIN 								// 
    PFFD           	: TIME := T#5S;       		// Feedback failure delay
    PTDH           	: TIME := T#5S;        	  	// Transit delay low to high
    PTDL           	: TIME := T#5S;       		// Transit delay high to low
    PSTO           	: BOOL;               		// Output YH and YL  constant on.
	PTTO			: TIME := T#2000MS;			// PULS output open YH
	PTTC			: TIME := T#2000MS;			// PULS output close YL
	PAOF			: INT  := 0;				// Parameter action on fault.
	PFT				: INT  := 3;				// Parameter feedback type
	PSUS			: INT  := 0;				// Parameter Template Startup State 
	PSUM			: INT  := 0;				// Parameter for mode at startup
	PSLO			: INT  := 0;				// Parameter for setting local or outside mode
END_VAR

VAR_OUTPUT
	Y              : BOOL;                		// 
	YH             : BOOL;               		// Normal output to switch control element to high state
    YL             : BOOL;                		// Normal output to switch control element to low state
    YF             : BOOL;                		// Control element fault
    BCH            : BOOL;               		// Binary status confirmed high
    BCL            : BOOL;                		// Binary status confirmed low
	BS             : BOOL;                		// Binary status safeguarding
	BB             : BOOL;                		// Binary status blocked
	BU             : BOOL;               		// Binary status suppressed
    BA             : BOOL;               		// Binary status automatic mode
	BO             : BOOL;                		// 
   // BM             : Bool := true;        	// Binary status manual mode    
   // BD             : Bool;                	// Binary status disabled
    YFI            : INT;               		// Fault information
END_VAR

VAR RETAIN
	
	sbBA           		 : BOOL;               	// Binary status automatic mode, RETAINED for prevstate.

END_VAR


VAR
	siState       		 : INT;                 // State of controlled element
    siNextState   		 : INT;                 // Next state of controlled element
	
	sbLA				: BOOL;					// Set auto variable
	sbLM				: BOOL;					// Set manual variable
	
	OS_FB				: BOOL;					// HMI Force block
	OS_FU				: BOOL;					// HMI Force supress
	OS_XLM				: BOOL;					// HMI Set low
	OS_XHM				: BOOL;					// HMI Set high
	
	TimerTransLow		: fbTimer;				// Timer trans low error
	TimerTransHigh		: fbTimer;				// Timer trans high erreor
	TimerFeedbackLow	: fbTimer;				// Timer no feedback low error
	TimerFeedbackHigh	: fbTimer;				// Timer no feedback high error
	OutputPulsHigh		: TP;
	OutputPulsLow		: TP;
	
	
	sbYF            : BOOL;						// Output fault variable
	sbBUpos			: BOOL;						// Binary supressed posetive flank variable
	sbBUneg			: BOOL;						// Binary supressed negative flank variable
	
	siFBlastvalue	: INT;						// 
END_VAR

VAR_TEMP

	tbHighCommand  		: BOOL;                 // High command
    tbLowCommand   		: BOOL;                 // Low Command
	tbOutsideLocal		: BOOL;					// Interlock of starting object when in local mode
	
	// INPUTS
	tbXGH            : BOOL;                	// eXternal Feedback Position High variable
    tbXGL            : BOOL;                	// eXternal Feedback Position Low variable
    tbXH             : BOOL;                	// eXternal Switch to Position High - in automatic mode variable
    tbXL             : BOOL;                	// eXternal Switch to Position Low - in automatic mode variable
	tbXOH            : BOOL;               		// eXternal Switch to Position High - In outside mode variable
	tbXOL            : BOOL;               		// eXternal Switch to Position LOW - In outside mode variable
	tbXF             : BOOL;                 	// eXternal Fault variable
	tbLSH            : BOOL;               		// Lock Safeguard High variable 
	tbLSL            : BOOL;               		// Lock Sagefuard Low variable 
	tbFSH            : BOOL;                	// Force Safeguarding High
    tbFSL            : BOOL;                	// [Priority] Force Safeguarding Low
    tbFDH            : BOOL;              		// Force Disable High
    tbFDL            : BOOL;             		// [Priority] Force Disable Low
	tbFB             : BOOL;             		// Force Blocking variable
	tbFU             : BOOL;					// Force Supression variable
	tbLA             : BOOL;               		// Lock Auto variable
	tbLM             : BOOL;               		// Lock Manuell variable
	tbLO             : BOOL;               		// Lock Outside
	
	
	// OUTPUTS
	tbY             : BOOL;                		// Output
	tbYH            : BOOL;               		// Normal output to switch control element to high state
    tbYL            : BOOL;                		// Normal output to switch control element to low state    
    tbBCH           : BOOL;               		// Binary status confirmed high
    tbBCL           : BOOL;                		// Binary status confirmed low
	tbBS            : BOOL;                		// Binary status safeguarding
	tbBB            : BOOL;                		// Binary status blocked
	tbBU            : BOOL;               		// Binary status supressed
	tbBO            : BOOL;                		// Binary status outside
	tiYFI			: INT;						// FAULT REGISTER
	
END_VAR

VAR CONSTANT
	ciInitState         : INT := 0;             // [FSM] Initial State of Control Element
    ciLow               : Int := 1;             // [FSM] Control Element in Low state
    ciTransitHigh       : Int := 2;             // [FSM] Control Element in transit to High state
    ciHigh              : Int := 3;             // [FSM] Control Element in High state
    ciTransitLow        : INT := 4;             // [FSM] Control Element in transit to Low state
	
	ciNoFault           : INT := 0;                  // [FAULT] No Fault Indication
    ciFeedbackFaultHigh : Int := 1;             // [FAULT] Feedback Fault
    ciFeedbackFaultLow  : Int := 2;             // [FAULT] Feedback Fault
    ciTransitHighFault  : Int := 3;             // [FAULT] Transit High Fault
    ciTransitLowFault   : INT := 4;             // [FAULT] Transit Low Fault
	ciExternalFault		: INT := 5;				// [FAULT] External fault
	ciConflictFault		: INT := 6;				// [FAULT] Conflict fault (Safeguard and blocking)
	ciSafeguardFault	: INT := 7;				// [FAULT] [Priority] Safeguard fault (No feedback while executing safeguard command)
	
	ciNoAction			: INT := 0;				// [PAOF] Parameter action on fault - No action
	ciClose				: INT := 1;				// [PAOF] Parameter action on fault - Closed action
	ciOpen				: INT := 2;				// [PAOF] Parameter action on fault - Open action
	
	ciNoFeedback		: INT := 0;				// [PFT] Parameter feedback mode - No feedback
	ciHighFeedback		: INT := 1;				// [PFT] Parameter feedback mode - High feedback
	ciLowFeedback		: INT := 2;				// [PFT] Parameter feedback mode - Low feedback
	ciFullFeedback		: INT := 3;				// [PFT] Parameter feedback mode - Full feedback
	
	ciStartupClosed		: INT := 0;				//
	ciStartupOpen		: INT := 1;
	ciStartupFeedback	: INT := 2;
	
	ciModeStartupManual		: INT := 0;			// Sets the mode of the block at startup
	ciModeStartupAuto		: INT := 1;			// Sets the mode of the block at startup
	ciModeStartupPrev		: INT := 2;			// Sets the mode of the block at startup
	
	ciModeLocal				: INT := 0;			// Parameter for setting local mode
	ciModeOutside			: INT := 1;			// Parameter for setting outside mode
END_VAR

//INFO, COPYRIGHT MANGOIPA GROUP INC
//SBV function block


//Populate Temporaries and preset outputs

tbXGH 									:= XGH;
tbXGL 									:= XGL;    
tbXH									:= XH;            
tbXL									:= XL;   
tbXOH									:= XOH;     
tbXOL									:= XOL;           
tbXF									:= XF;            
tbLSH									:= LSH;           
tbLSL									:= LSL;           
tbFSH									:= FSH;           
tbFSL									:= FSL;            
tbFDH									:= FDH;            
tbFDL									:= FDL;            
tbFB									:= FB;            
tbFU									:= FU;            
tbLA									:= LA;              
tbLM									:= LM;             
tbLO									:= LO;       

// Timers
TimerTransLow();													// Timer for transition to low fault
TimerTransHigh();													// Timer for transition to high fault
TimerFeedbackLow();													// Timer for no feedback low fault
TimerFeedbackHigh();												// Timer for no feedback high fault
OutputPulsHigh();										 			// Timer for puls YH
OutputPulsLow();													// Timer for puls YL

//Timer parameters (should be behind a restart/startup function))
TimerTransLow.PTDH						:= PTDH;
TimerTransHigh.PTDH 					:= PTDL;
TimerFeedbackLow.PTDH					:= PFFD;
TimerFeedbackHigh.PTDH					:= PFFD;
OutputPulsHigh.PT						:= PTTO;
OutputPulsLow.PT						:= PTTC;


// Handle external faults, subject to supression
IF (tbXF AND NOT tbFU) THEN
	tiYFI 								:= ciExternalFault;
END_IF

// Handle High output puls YH / YL
IF NOT (siState = ciTransitHigh) THEN
	OutputPulsHigh.IN 					:= FALSE;
END_IF

IF NOT (siState = ciTransitLow) THEN
	OutputPulsLow.IN 					:= FALSE;
END_IF


// MODECONTROLL
// Mode Control - AUTO/MAN
IF tbLM AND NOT sbLM  THEN
    sbBA                       			:= FALSE;					// Manual mode, BA = 0
ELSIF tbLA AND NOT sbLA THEN
    sbBA                       			:= TRUE; 	    			// Auto mode posetive edge,	BA = 1
END_IF;
	
sbLA 									:= tbLA;					// Retrigger posetive edge for Mode Control.
sbLM 									:= tbLM;					// Retrigger posetive edge for Mode Control.

// Mode Controll - Outside/Local mode.
IF tbLO THEN		
	tbBO 								:= TRUE;					// Sets status outside and force off auto-mode
	sbBA 								:= FALSE;	
	
	CASE PSLO OF													// Case for Parameter for setting local/outside
	ciModeLocal:	
		tbOutsideLocal				    := TRUE;					// Switches the block between High and Low in local mode from XGH/XGL
		IF tbXGH THEN	
			siState 					:= ciHigh;
		ELSIF tbXGL THEN			
			siState					    := ciLow;
		END_IF
				
	ciModeOutside: 													// If in outside mode, XOH/XOL will controll the block
	tbOutsideLocal 						:= FALSE;
	//
	END_CASE
ELSE
	tbBO 								:= FALSE;							
END_IF	

// SAFEGUARDING (Stod tidligere over modecontroll.)
// Handle lock safeguard mode, subject to blocking
IF (tbLSL AND NOT tbFB) THEN
	sbBA 								:= FALSE;					// Set mode to manual
ELSIF (tbLSH AND NOT tbFB) THEN
	sbBA 								:= FALSE;					// Set mode to manual
END_IF

// Handling safeguarding BS status, triggered by any Safeguarding
IF (tbLSH OR tbLSL OR tbFSH OR tbFSL) THEN
	tbBS 								:= TRUE;
ELSE
	tbBS 								:= FALSE;
END_IF

// Handling blocking BB status
IF (tbFB OR OS_FB) THEN
	tbBB 								:= TRUE;
ELSE
	tbBB 								:= FALSE;
END_IF

//Blocking blocks safeguard and disable transition modes
IF tbBB THEN
	tbLSL 								:= FALSE;
	tbLSH							    := FALSE;
	tbFSL 								:= FALSE;
	tbFSH 								:= FALSE;
	tbFDH 								:= FALSE;
	tbFDL 								:= FALSE;
END_IF

// Handle conlfict fault when safeguarding and blocking. ( Stod tidligre under low & high command)
IF (tbBS AND tbBB) THEN
	tiYFI 							    := ciConflictFault;
END_IF

// SUPRESSION
// Handling supression BU status ON/OFF
IF (tbFU OR OS_FU) THEN
	tbBU  								:= TRUE;	
ELSE
	tbBU 								:= FALSE;
END_IF

// Handles supression and PFT (Parameter feedback type)
IF tbBU AND NOT sbBUpos THEN
	siFBlastvalue 						:= PFT;						// Stores PFT before supression sets to "no feedback" on posetive edge
	PFT									:= ciNoFeedback;
END_IF

IF NOT tbBU AND sbBUneg THEN										// sets PFT to last value on negative edge
	PFT 								:= siFBlastValue;
END_IF

sbBUpos									:= tbBU;					// Posetive edge retrigger
sbBUneg 								:= tbBU;    				// Negative edge retrigger

//LOW AND HIGH COMMAND
//High and low commands evaluation (AUTO & MANUAL & OUTSIDE & LSL & LSH FDL & FDH
tbLowCommand                 		    := (tbXL AND sbBA) OR 										// Auto 
								 		   (OS_XLM AND NOT sbBA AND NOT tbBO) OR 					// Manuell (Triggered by XLM supressed by Auto & Outside mode)
								 		   (tbBO AND tbXOL AND NOT tbOutsideLocal) OR 				// Outside (Triggered by XOL if in not local outside mode)	
								 		   (tbLSL AND NOT tbFB) OR									// Lock Safeguard Low subject by blocking
								 		   (tbFSL AND NOT tbFB);									// Force safeguard Low subject by blocking
												

tbHighCommand                 			:= (tbXH AND sbBA) OR 										// Auto
								           (OS_XHM AND NOT sbBA AND NOT tbBO AND NOT tbBS) OR 		// Manuell (Triggered by XLM supressed by Auto & Outside mode
								           (tbBO AND tbXOH AND NOT tbOutsideLocal) OR 				// Outside (Triggered by XOL if in not local outside mode)
								           (tbLSH AND NOT tbFB) OR									// Lock Safeguard Low subject by blocking
								           (tbFSH AND NOT tbFB);									// Force safeguard Low subject by blocking
											

										   
// Handle force disable high command and low command
IF tbFDH AND NOT tbFB THEN
    tbHighCommand            			:= FALSE;   				//If FDH is true then erase high command, prevent transit to high
END_IF;

IF tbFDL AND NOT tbFB THEN
    tbLowCommand             			:= FALSE;   				//If FDL is true then erase low command, prevent transit to low
END_IF;

// Handle Force safeguard commands
IF tbFSL THEN
    tbHighCommand            			:= FALSE;
    tbLowCommand              			:= NOT tbXGL;    			// As long as FSL is true and not correct feedback, force transit to low
	
ELSIF tbFSH THEN													// I manuell skal den ha Y = 0 (lukka) etter FSL er ute. (Høgkant OS_XLH?)
    tbHighCommand             			:= NOT tbXGH;   			// As long as FSH is true and not correct feedback, force transit to high
    tbLowCommand              			:= FALSE;	
// I manuell skal den ha Y = 1 (lukka) etter FSL er ute.
END_IF;


// Handle parameter action on fault
IF sbYF THEN
	CASE PAOF OF 
		ciNoAction:									   			     // No action on fault			
			sbYF 						:= sbYF;		
		ciClose:													 // Close
			tbLowCommand 				:= TRUE;		
		ciOpen:														 // Open
			tbHighCommand 				:= TRUE;		
	END_CASE	
END_IF


// Handle parameter feedbacks - Sets the mode of feedback
CASE PFT OF
	ciNoFeedback:
		tbXGH 							:= (siState = ciHigh) OR (siState = ciTransitHigh);	// If no feedback mode, the state sets the XGH/XGL direct			
		tbXGL 							:= (siState = ciLOW)  OR (siState = ciTransitlow);
	ciHighFeedback:
		tbXGL 							:= (siState = ciLOW)  OR (siState = ciTransitlow);	// If no High feedback, the transition or low state sets XGL direct
	ciLowFeedback:
		tbXGH 							:= (siState = ciHigh) OR (siState = ciTransitHigh);	// If no High feedback, the transition or high state sets XGH direct
	ciFullFeedback:
		tbXGH 							:= tbXGH;
		tbXGL := tbXGL;
END_CASE;


//Determine next state
IF tbHighCommand THEN
    siNextState              		    := ciHigh;
ELSIF tbLowCommand THEN
    siNextState              		    := ciLow;
End_If;


//Tilstandsmaskina 
CASE siState OF 
	//INIT STATE
	ciInitState:														// Initial state, sets some parameters for startup
	
	CASE PSUM OF														// Sets the Statup mode.
			ciModeStartupManual		: 
				sbBA 					:= FALSE;
							
			ciModeStartupAuto		: 
				sbBA 					:= TRUE;	
		
			ciModeStartupPrev		: 
				sbBA 					:= sbBA;
	END_CASE
	
	//Sets the startup state of the block - Parameter Template Startup State
	CASE PSUS OF														
		ciStartupClosed		:  
			siState := ciLow;
			
		ciStartupOpen		:  
			siState := ciHigh;
			
		ciStartupFeedback	:  											// If feedback state, XGL/XGH determines the start state of the block
			IF tbXGH THEN
				siState					:= ciHigh;
			ELSIF XGL THEN
				siState 				:= ciLow;		
			END_IF
	END_CASE
	
	// Case for handling next state
	CASE siNextState OF
		ciHigh: 
			siState						:= ciTransitHigh;
			
		ciLow :	
			siState 		 			:= ciTransitLow;		
	END_CASE	
	
	// LOW STATE 
	ciLow:	
	
		IF (NOT tbXGL OR tbXGH) THEN									// Faulthandling if no feedback detected	
		    TimerFeedbackLow.X := TRUE;
	
            IF TimerFeedbackLow.Y THEN									// Starts the timer if missing feedback detected
                tiYFI           		:= ciFeedbackFaultLow;
            END_IF;
        ELSE
            TimerFeedbackLow.X := FALSE;								// Resets timer if feedback returns
        End_If;

        CASE siNextState OF												// Sets the next state
            ciHigh :                
                siState      		 	:= ciTransitHigh;
        END_CASE;
	
	// TRANSIT HIGH STATE	
	ciTransitHigh:
		
		TimerTransHigh.X 				:= TRUE;						// Sets timer for allowed time before feedback
		OutputPulsHigh.IN 			    := TRUE;						// Sets timer for puls output
				
		IF tbXGH THEN													// Feedback detected, resets timers and changes state
			TimerTransHigh.X 		    := FALSE;
			siState           		    := ciHigh;
		END_IF			
	
		IF (TimerTransHigh.Y) THEN										// Handles no feedback fault
			tiYFI						:= ciTransitHighFault;
		END_IF
		
		CASE siNextState OF												// Changes state 
            ciLow :                
                siState     		    := ciTransitLow;
        End_Case;
		
	ciHigh:
	//HIGH STATE	
	    IF (NOT tbXGH OR tbXGL) THEN									// Faulthandling when no feedback			
            TimerFeedbackHigh.X 		:= TRUE;						// Starts timer when no feedback
			
            IF TimerFeedbackHigh.Y THEN									// Faulthandling of timer
                tiYFI           		:= ciFeedbackFaultHigh;
            END_IF;
        ELSE
            TimerFeedbackHigh.X 		:= FALSE;						// Resets timer if feedback returns
        End_If;
		
        CASE siNextState OF												// Changes states 
            ciLow :
                siState       		  	:= ciTransitLow;
        End_Case;
	
	ciTransitLow:
	//TRANSIT LOW STATE
		TimerTransLow.X 				:= TRUE;						// Starts timer for transit 
		OutputPulsLow.IN 				:= TRUE;						// Starts timer for pulse YL
	
		IF tbXGL THEN	
			TimerTransLow.X 			:= FALSE;						// Reset timer if feedback
			siState          			:= ciLOW;						// Changes from transit to Low 
		END_IF
		
			IF (TimerTransLow.Y) THEN									// Faulthandling if no feedback
				tiYFI					:= ciTransitLowFault;	
			END_IF
		
		CASE siNextState OF												// Changes states 
            ciHigh :                
                siState      		 	:= ciTransitHigh;
        End_Case;	

END_CASE

// Safeguard fault if safeguard and no feedback fault
IF (tbBS AND ((tiYFI = ciFeedbackFaultHigh) OR (tiYFI = ciFeedbackFaultLow))) THEN
	tiYFI 							    := ciSafeguardFault;
END_IF;

// FAULT handling
sbYF 									:= (tiYFI > ciNoFault);

//Handle supression of YF
IF tbBU THEN
	sbYF							    := FALSE;
END_IF


//Write to output //TATT FRA OLAV DIREKTE
Y										:= 	(siState = ciTransitHigh) OR ((siState = ciHigh));
YH                            			:=	OutputPulsHigh.Q OR (PSTO AND (siState = ciTransitHigh)) ;
YL                           			:= 	OutputPulsLow.Q OR (PSTO AND (siState = ciTransitLow)) ;
BA										:= 	sbBA;
BU										:=  tbBU;
YF                           			:= 	(sbYF);
YFI										:=  tiYFI;
BCH                          			:= 	(siState = ciHigh) AND tbXGH AND NOT tbXGL;
BCL                         			:= 	(siState = ciLow) AND tbXGL AND NOT tbXGH;
BS										:=  tbBS;

//Write to HMI

END_FUNCTION_BLOCK

// Device/Application/test_SFC
PROGRAM test_SFC
VAR
END_VAR

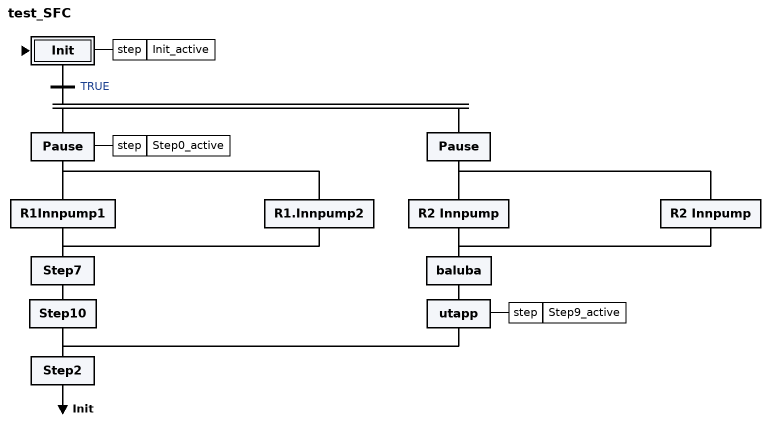
INITIAL_STEP Init:
    Init_active(N);  // step action
END_STEP
TRANSITION FROM Init TO (Pause, Pause)
    := TRUE;
END_TRANSITION
STEP Pause:
    Step0_active(N);  // step action
END_STEP
// no transition between Pause and R1Innpump1
// no transition between Pause and R1.Innpump2
STEP R1Innpump1:
END_STEP
// no transition between R1Innpump1 and Step7
STEP R1_Innpump2:  // name as stored: R1.Innpump2
END_STEP
// no transition between R1.Innpump2 and Step7
STEP Step7:
END_STEP
// no transition between Step7 and Step10
STEP Step10:
END_STEP
// no transition between Step10 and Step2
STEP Pause:
END_STEP
// no transition between Pause and R2 Innpump
// no transition between Pause and R2 Innpump
STEP R2_Innpump:  // name as stored: R2 Innpump
END_STEP
// no transition between R2 Innpump and baluba
STEP R2_Innpump:  // name as stored: R2 Innpump
END_STEP
// no transition between R2 Innpump and baluba
STEP baluba:
END_STEP
// no transition between baluba and utapp
STEP utapp:
    Step9_active(N);  // step action
END_STEP
// no transition between utapp and Step2
STEP Step2:
END_STEP
// no transition between Step2 and Init
// branch label varInnpumpOK
// branch label VarInnpumpok2

ACTION Init_active:

END_ACTION

END_PROGRAM

// Device/Application/tmReactor1
FUNCTION_BLOCK tmReactor1
VAR_INPUT
//  	PP00_LT01_AHH				: BOOL;					// Mottaktstank nivåmåler
//  	PP00_LT01_ALL				: BOOL;					// Mottaktstank nivåmåler
//  	PP00_LS02					: BOOL;					// Inngang for vippe i mottakstank HIGH HIGH
//  	PP00_LS01					: BOOL;					// Inngang for vippe i mottakstank LOW LOW 		
//  	PP01_LT01					: BOOL;					// Reaktor 1 nivå¨måler
END_VAR

VAR_OUTPUT	

END_VAR

VAR_TEMP	
	//Innputs
	tbXE							: BOOL;
	tblt_Mottakstank_AHH			: BOOL;						// ER Høg om nivå er over tillatt innpumping
	tblt_Mottakstank_ALL			: BOOL;						// ER Høg om nivå er over tillatt innpumping
	tbls_hog						: BOOL;
	tbls_lav						: BOOL;	

	//Output
	tbPause						: BOOL;							//
	tbInnpumping 				: BOOL;
	tbInnpumping_Pause			: BOOL;
	tbReaksjon 					: BOOL;
	tbSedementering 			: BOOL;
	tbUttapping					: BOOL;
	
END_VAR


VAR
	siState						: INT;		
	sitest 						: INT;
	InnpumpingTimer				: fbTimer;
	ReaksjonTimer				: fbTimer;
	SedimenteringTimer			: fbTimer;
	UttappingTimer				: fbTimer;
	
	Pause						: fbPause;
	Innpumping					: fbInnpumping;
END_VAR


VAR CONSTANT
	ciInit				     	: INT := 0;		
	ciPause			     		: INT := 1;						
	ciInnpumping 		     	: INT := 2;		
	ciInnpumping_Pause			: INT := 3;		
	ciReaksjon 			     	: INT := 4;		
	ciSedementering 		    : INT := 5;		
	ciUttapping			 	    : INT := 6;	
		
END_VAR

//Tilstandsmaskin som styrer 1 reaktor.

 //tblt_Mottakstank_AHH			:= PP00_LT01_AHH;
 //tblt_Mottakstank_ALL			:= PP00_LT01_ALL;
 //tbls_hog						:= PP00_LS02;
 //tbls_lav						:= PP00_LS01;

//Timer
InnpumpingTimer();
ReaksjonTimer();
SedimenteringTimer();	
UttappingTimer();

//Setter tid til timere - Må endres til GVB på ett tidspunkt.
InnpumpingTimer.PTDH				:= GVL_Sekvenstider.TidInnpumpingMaks;
ReaksjonTimer.PTDH 					:= GVL_Sekvenstider.TidReaksjon;
SedimenteringTimer.PTDH				:= GVL_Sekvenstider.TidSedimentering;	
UttappingTimer.PTDH					:= GVL_Sekvenstider.TidUttapping;


CASE siState OF
	ciInit:
		//Setter timere 
		siState 					:= ciPause;
		
	ciPause	:	
		tbPause 					:= TRUE;
		
		//Reset av timers	
		InnpumpingTimer.X				:= FALSE;
		ReaksjonTimer.X					:= FALSE;
		SedimenteringTimer.X			:= FALSE;	
		UttappingTimer.X				:= FALSE;	
		
		//Pause();
		
		IF GVL_TM.PauseReaktor1OK THEN	// forrigling mot R2
			siState 				:= ciInnpumping;
		END_IF	
	
	 
	ciInnpumping :	
	//	
		tbInnpumping 						:= TRUE;		
		
		//Innpumping();
				
		IF (GVL_TM.InnpumpingReaktor1OK) THEN
			siState 						:= ciReaksjon;
		END_IF
				
		
// 		InnpumpingTimer.X					:= TRUE;
// 		IF (PP01_LT01 OR InnpumpingTimer.Y ) THEN									// Eller timer
// 			siState 						:= ciReaksjon;
// 		END_IF
// 		
// 		IF (PP00_LT01_ALL OR PP00_LS01) THEN
// 			siState := ciInnpumping_Pause;
// 		END_IF
	
// 	ciInnpumping_Pause: 	
// 	//	
// 		tbInnpumping_Pause 					:= TRUE;
// 		IF (tblt_Mottakstank_AHH OR tbls_hog ) THEN								
// 			siState 						:= ciInnpumping;
// 		END_IF
// 		
// 		IF InnpumpingTimer.Y THEN
// 			siState 						:= 	ciReaksjon;
// 		END_IF
		
	ciReaksjon: 	
	//	
		tbReaksjon 							:= TRUE;
		ReaksjonTimer.X						:= TRUE;
		
		IF (ReaksjonTimer.Y) THEN
			siState 						:= ciSedementering;
		END_IF
		
	ciSedementering : 	
	//	
		tbSedementering 					:= TRUE;
		SedimenteringTimer.X				:= TRUE;
		
		IF (SedimenteringTimer.Y) THEN
			siState 						:= ciUttapping;
		END_IF
		
	ciUttapping	: 			
	//	
		tbUttapping 						:= TRUE;
		UttappingTimer.X					:= TRUE;
		
		IF (UttappingTimer.Y) THEN
			siState 						:= ciPause;
		END_IF

END_CASE




//Outputs
GVL_TM.Pause1						:= tbPause;
GVL_TM.Innpumping1 					:= tbInnpumping;
GVL_TM.Innpumping_Pause1		 		:= tbInnpumping_Pause;
GVL_TM.Reaksjon1 					:= tbReaksjon;
GVL_TM.Sedementering1 				:= tbSedementering;
GVL_TM.Uttapping1					:= tbUttapping;

END_FUNCTION_BLOCK

// Device/Application/Utrekningar
PROGRAM Utrekningar
VAR
	sjekk	: 			REAL;
END_VAR


// Beregne frå nivå til volum reaktor 1
VolumReaktor(Height := GVL_R1.Nivaa, Volum => GVL_R1.Volum);


// Beregne frå nivå til volum reaktor 2
VolumReaktor(Height := GVL_R1.Nivaa, Volum => GVL_R1.Volum);

END_PROGRAM

// Device/Application/Common_Functions/CommonFunctions
PROGRAM CommonFunctions
VAR
	Utrekning 				: fbCalculations;
	SivbedRotation 		    : fbSivbedRotation;
	Databehandling			: fbDataprocessing;
	O_Map					: Output_Mapping;
	HoyB					: fbHighload;
	ProcessedWater					: fbProcessedWater;
END_VAR

Utrekning(); // fbCalculations
SivbedRotation(
    X := GVL_Rest.PulseCoutner,
    X2 := GVL_Rest.GangerPrSivBed,
    XE1 := GVL_Rest.ActiveCelle1,
    XE2 := GVL_Rest.ActiveCelle2,
    XE3 := GVL_Rest.ActiveCelle3,
    XE4 := GVL_Rest.ActiveCelle4); // fbSivbedRotation
GVL_Rest.siSivState := SivbedRotation.Y;
// Bool input frå GVL
Databehandling(
    X0 := GVL_Outputs.PP01_PS01_Y,
    X1 := GVL_Outputs.PP02_PS01_Y,
    X2 := GVL_Outputs.PA01_BL01_Y,
    X3 := GVL_Outputs.PA02_BL01_Y,
    X4 := GVL_Outputs.CH00_PH01_Y,
    X5 := GVL_Outputs.CH00_PH02_Y,
    X6 := GVL_Outputs.RET_PHUS_Y,
    X7 := GVL_Outputs.DRE_PHUS_Y); // fbDatabehandling
GVL_Rest.PP02_PS01_Tottid := Databehandling.Y1;
GVL_Rest.PA01_BL01_Tottid := Databehandling.Y2;
GVL_Rest.PA02_BL01_Tottid := Databehandling.Y3;
GVL_Rest.CH00_PH01_Tottid := Databehandling.Y4;
GVL_Rest.CH00_PH02_Tottid := Databehandling.Y5;
GVL_Rest.RET_PHUS_Tottid := Databehandling.Y6;
GVL_Rest.DRE_PHUS_Tottid := Databehandling.Y7;
// Tider output til GVL
GVL_Rest.PP01_PS01_Tottid := Databehandling.Y0;
O_MAP(); // OUTPUT_MAPPING
HoyB(X := GVL_REST.MottakstankNivaa, PXR := GVL_REST.LimitHoybelastning); // fbHighload
GVL_Rest.HoyBelastning := HoyB.Y;
GVL_Rest.AntattTilrenning := HoyB.YG;
ProcessedWater(X1 := GVL_R1.DeltaKubikkDrenert, X2 := GVL_R2.DeltaKubikkDrenert); // fbProcessedWater
GVL_Rest.TotaltBehandlaVatn := ProcessedWater.Y1;
GVL_Rest.TotYear := ProcessedWater.Y2;
GVL_Rest.TotMonth := ProcessedWater.Y3;
GVL_Rest.TotWeek := ProcessedWater.Y4;
GVL_Rest.TotDay := ProcessedWater.Y5;
GVL_Rest.LastYear := ProcessedWater.Y6;
GVL_Rest.LastMonth := ProcessedWater.Y7;
GVL_Rest.LastWeek := ProcessedWater.Y8;
GVL_Rest.LastDay := ProcessedWater.Y9;

END_PROGRAM

// Device/Application/Function blocks/fbSivbedRotation
FUNCTION_BLOCK fbSivbedRotation
VAR_INPUT
	X					: BOOL;		// Normal functuon input, pulsed each time a reactor goes throigh slamtapping sequence
	XE1					: BOOL;		// Enable for rotation sivbed 1
	XE2					: BOOL;		// Enable for rotation sivbed 2
	XE3					: BOOL;		// Enable for rotation sivbed 3
	XE4					: BOOL;		// Enable for rotation sivbed 4
END_VAR

VAR_INPUT RETAIN
	X2					: INT;		// Input interger value that decides how many slamcycels one sivbed has before it rotates
END_VAR

VAR_OUTPUT
	Y					: SINT;		// Output integer value that outputs wich sivbed is currently in rotation
END_VAR

VAR
	SiSivBed			: SINT;
	siTeller			: INT;
	sbPulseCounter		: BOOL;
END_VAR

VAR CONSTANT
	ciInit				: SINT := 0;
	ciCelle1			: SINT := 1;
	ciCelle2			: SINT := 2;
	ciCelle3			: SINT := 3;
	CiCelle4			: SINT := 4;
END_VAR

//Handles the rotation of Sivebed, based on amount sivebed is used, counted from Reaktors



//Handle count of sivbed 
IF (X AND NOT sbPulseCounter) THEN	
	siTeller := siTeller + 1;			// Increase count by 1;
END_IF

sbPulseCounter := X;


IF (siTeller > X2) THEN
	siSivBed := siSivBed + 1;
	siTeller := 0;
END_IF


CASE (SiSivBed) OF
			
			ciInit:	
			
				SiSivBed := ciCelle1;
			
			ciCelle1:			
			// Sender vidare dersom Sivbed er tatt ut av drift				
				IF NOT (XE1) THEN
					SiSivBed := ciCelle2;
				END_IF
						
			ciCelle2:			
			// Sender vidare dersom Sivbed er tatt ut av drift	
				IF NOT (XE2) THEN
					SiSivBed := ciCelle3;
				END_IF
			
			ciCelle3:		
			// Sender vidare dersom Sivbed er tatt ut av drift	
				IF NOT (XE3) THEN
					SiSivBed := ciCelle4;
				END_IF
			
			ciCelle4:		
			// Sender vidare dersom Sivbed er tatt ut av drift		
				IF NOT (XE4) THEN
					SiSivBed := ciCelle1;
				END_IF
		
ELSE
	SiSivBed := ciCelle1;		
END_CASE

// OUTPUT
Y			:= siSivbed;

END_FUNCTION_BLOCK

// Device/Application/Function blocks/fbDatabehandling
FUNCTION_BLOCK fbDatabehandling
VAR_INPUT
	X0	: BOOL;
	X1	: BOOL;
	X2	: BOOL;
	X3	: BOOL;
	X4	: BOOL;
	X5	: BOOL;
	X6	: BOOL;
	X7	: BOOL;

END_VAR
VAR_OUTPUT

	Y0 : TIME;	
	Y1 : TIME;	
	Y2 : TIME;	
	Y3 : TIME;	
	Y4 : TIME;	
	Y5 : TIME;	
	Y6 : TIME;
	Y7 : TIME;	
	
END_VAR
VAR
	PP01_PS01		: fbCAC;	// Innpumpe nr 1
	PP02_PS01		: fbCAC;	// Innpumpe nr 2
	PA01_BL01		: fbCAC;	// Blåser 1
	PA02_BL01		: fbCAC;	// Blåser 2
	CH00_PH01		: fbCAC;	// Doseringspumpe 1
	CH00_PH02		: fbCAC;	// Doseringspumpe 2
	RET_PHUS		: fbCAC;	// Return på Pumpehus og sivbed
	DRE_PHUS		: fbCAC;	// Til resepient Pumpehus
END_VAR

// Time teller for innpumpe Nr 1
PP01_PS01();
PP01_PS01.X := X0;
Y0 := PP01_PS01.Tid;

// Time teller for innpumpe Nr 1
PP02_PS01();
PP02_PS01.X := X1;
 Y1 := PP02_PS01.Tid;

// Time teller for blåser 1
PA01_BL01();
PA01_BL01.X := X2;
Y2 := PA01_BL01.Tid;

// Time teller for blåser 2
PA02_BL01();
PA02_BL01.X := X3;
Y3 := PA02_BL01.Tid;

// Time teller for doseringspumpe 1
CH00_PH01();
CH00_PH01.X	:= X4;
Y4 := CH00_PH01.Tid;

// Time teller for doseringspumpe 2
CH00_PH02();
CH00_PH02.X	:= X5;
Y5 := CH00_PH02.Tid;

// Time teller for return på sivbed
RET_PHUS();
RET_PHUS.X := X6;
Y6 := RET_PHUS.Tid;

// Time teller for drenering mot resepient på sivbed
DRE_PHUS();
DRE_PHUS.X := X7;
Y7 := DRE_PHUS.Tid;

END_FUNCTION_BLOCK

// Device/Application/Function blocks/fbCAC
FUNCTION_BLOCK fbCAC
VAR_INPUT
	X			: BOOL;
END_VAR
VAR_OUTPUT
	Y  				: BOOL;			// Limit violation	

	Tid			: TIME;
	Dager		: INT;
	Timer		: INT;
	Minutt		: INT;
	Sekund		: INT;
	
	TotTimer	: LINT;
END_VAR
VAR
	stTimeOn 		: TIME;
	stTimeOff 		: TIME;
	sbDelayBlock    : BOOL;			//Beskyttelse
	sbY				: BOOL;
	sbX				: BOOL;
	
	Gangtid			: TIME;
END_VAR
VAR RETAIN
	TotalTid		: TIME;
END_VAR

VAR_TEMP
	
	// TEMP INPUTS
	tbX				: BOOL;	
	
	ttNow 			: TIME;
	ttTimeOn 		: TIME;
	ttTimeOff 		: TIME;
	
	tiMillis		: LINT;
	
	tiSekund		: LINT;
	tiMinutt		: LINT;
	tiTimer			: LINT;
	tiDays			: LINT;
	tiTotTimer		: LINT;
	tiRestMillis	: LINT;
	

END_VAR

VAR CONSTANT
	cliMillis2Days : LINT := 86400000;
	cliMillis2Hours : LINT := 3600000;
	cliMillis2Minutes : LINT := 60000;
	cliMillis2Seconds : LINT := 1000;

END_VAR

// ***************************************************************************************
// Copyright: Peter Søreide Skaar, Roar Bøyum, Vegard Aven Ullebø [2024]
// All rights reserved.

// This code was developed as part of a Bachelor's thesis conducted for Renasys AS 
// and Sunnfjord Kommune. 

// Unauthorized reproduction, distribution, or modification of this code, in whole 
// or in part, is strictly prohibited without the express permission of the copyright 
// holder.
// ***************************************************************************************


// INPUTS
tbX 								:= X;

// ttNow gets PLC time
ttNow 								:= TIME();							

// ttTime teller tida
ttTimeON 							:= ttNow - stTimeOn;
ttTimeOff 							:= ttNow - stTimeOff;

// OnDelay
IF tbX THEN
	sbDelayBlock 					:= FALSE;

	sbY 							:= TRUE;
	Gangtid := (ttTimeON-ttTimeOFF);	

ELSE	
	sbDelayBlock 					:= TRUE;
	stTimeOn  						:= ttNow;
END_IF;

// OffDelay
IF NOT tbX AND sbDelayBlock THEN
	
	sbY 							:= FALSE;
					
ELSE
	stTimeOff  							:= ttNow;	
END_IF;

// Negativ flanke på X, køyrest ein gong og tid lagrast til totaltida.

IF NOT tbX AND sbX THEN
	TotalTid := TotalTid + Gangtid;
	
	// Conversion of time from TIME variable to DAYS / HOURS / MINUTES / SECONDS
	
	tiMillis 		:= TIME_TO_LINT(TotalTid);
	
	tiDays 			:= tiMillis / cliMillis2Days;
	tiRestMillis 	:= tiMillis - (tiDays * CliMillis2Days);
	
	tiTotTimer		:= tiMillis / cliMillis2Hours;
	
	tiTimer := tiRestMillis / cliMillis2Hours;
	tiRestMillis 	:= tiRestMillis - (tiTimer * CliMillis2Hours);
	
	tiMinutt := tiRestMillis / cliMillis2Minutes;
	tiRestMillis 	:= tiRestMillis - (tiMinutt * CliMillis2Minutes);
	
	tiSekund := tiRestMillis / cliMillis2Seconds;
	tiRestMillis 	:= tiRestMillis - (tiSekund * CliMillis2Seconds);
	
END_IF

// Negativ flank retrigger
sbX := tbX;


// OUTPUTS
Y 										:= sbY;
Tid										:= TotalTid;
Dager									:= LINT_TO_INT(tiDays);
Timer									:= LINT_TO_INT(tiTimer);
Minutt									:= LINT_TO_INT(tiMinutt);
Sekund									:= LINT_TO_INT(tiSekund);
TotTimer								:= tiTotTimer;

END_FUNCTION_BLOCK

// Device/Application/Function blocks/Output_Mapping
FUNCTION_BLOCK Output_Mapping
VAR_INPUT
END_VAR
VAR_OUTPUT
END_VAR
VAR
END_VAR


// Handle all blower PA01_BL01 run signal to one output
GVL_Outputs.PA01_BL01_Y := GVL_R1.Pause_PA01_BL01 OR GVL_R1.Innpumping_PA01_BL01 OR GVL_R1.Reaksjon_PA01_BL01;

// Handle all blower PA02_BL01 run signal to one output


// Handle all matepumpe 1 run signals to one output
GVL_Outputs.PP01_PS01_Y := GVL_R1.PP01_PS01_Y OR GVL_R2.PP01_PS01_Y;

// Handle all matepumpe 2 run signals to one output
GVL_Outputs.PP02_PS01_Y := GVL_R1.PP02_PS01_Y OR GVL_R2.PP02_PS01_Y;

// Handle all sivcelle 1 valve open to one output
GVL_Outputs.PS00_VP01_Y := GVL_R1.PS00_VP01_Y OR GVL_R2.PS00_VP01_Y;

// Handle all sivcelle 2 valve open to one output
GVL_Outputs.PS00_VP02_Y := GVL_R1.PS00_VP02_Y OR GVL_R2.PS00_VP02_Y;

// Handle all sivcelle 3 valve open to one output
GVL_Outputs.PS00_VP03_Y := GVL_R1.PS00_VP03_Y OR GVL_R2.PS00_VP03_Y;

// Handle all sivcelle 4 valve open to one output
GVL_Outputs.PS00_VP04_Y := GVL_R1.PS00_VP04_Y OR GVL_R2.PS00_VP04_Y;

END_FUNCTION_BLOCK

// Device/Application/Function blocks/fbHighload
FUNCTION_BLOCK fbHighload
VAR_INPUT
	X						: REAL;

END_VAR

VAR_INPUT RETAIN
	PXR						: REAL;
END_VAR


VAR_OUTPUT
	Y						: BOOL;
	YG						: REAL;
END_VAR
VAR
	Timer					: fbTimer;
	sbY						: BOOL;
	srSample				: REAL;
	srLastSample			: REAL;
	srDelta					: REAL;
	trDelta					: REAL;
	
	FIFO					: ARRAY[1..ciArraySize] OF REAL;
	
	teller					: INT;
//END_VAR

//VAR_TEMP
	Sum						: REAL;
	Avarage					: REAL;
END_VAR

VAR CONSTANT
	SampleTime				: TIME		:= T#1M;
	crMottakstankBreidde	: REAL		:= 6.0;
	crMottakstankLengde		: REAL		:= 6.0;
	ciArraySize				: INT		:= 30;
END_VAR

//Measure over 30mins and calculates the avrage flow over 60mins


// Initialize timer
Timer();
Timer.PTDH 					:= SampleTime;

// Start timer
Timer.X 					:= TRUE;

// Saves sampled value each time timer goes true
IF (Timer.Y AND NOT sbY) THEN

	// Resetting sum
	SUM := 0;

	// Reads current value
	srSample				:= X;		
	srDelta					:= srSample - srLastSample;	
	trDelta 				:= srDelta * crMottakstankBreidde * crMottakstankLengde;
	
	// Protection against "Innpumping" negative trend.
	IF (trDelta < 0) THEN
		trDelta 			:= 0;
	END_IF
	
	
	// Moves all values in array 1 next	
	FOR teller := (ciArraySize - 1) TO 1 BY -1 DO
		FIFO[teller + 1]	:= FIFO[teller];
	END_FOR
	
	//Add into array
	FIFO[1] 				:= trDelta;
	
	// Store value
	srLastSample 			:= srSample;
	
	
	// Calculate the avarage delta across the FIFO 30min	
	FOR teller := 1 TO ciArraySize DO
		SUM 				:= SUM + FIFO[Teller];
	END_FOR	
	
	Avarage 				:= SUM / ciArraySize;
	
	// Calculates flow/hour
	YG 		:= Avarage *2;
	
	IF (YG > PXR) THEN
		Y 		:= TRUE;
	ELSE
		Y 		:= FALSE;
	END_IF
	
	IF (Y) THEN		
		// Endre sekvenstider		
		GVL_R1.SekvenstidReaksjon 		:= GVL_R1.SekvenstidReaksjonHoyg;
		GVL_R1.SekvenstidSedimentering 	:= GVL_R1.SekvenstidSedimenteringHoyg;
	ELSE
		// Vanlege sekvenstider		
		GVL_R1.SekvenstidReaksjon 		:= GVL_R1.SekvenstidReaksjonLav;
		GVL_R1.SekvenstidSedimentering 	:= GVL_R1.SekvenstidSedimenteringLav;				
	END_IF
	
	// Reset timer
	Timer.X 				:= FALSE;
END_IF


//Reset posetiv edge detection
sbY							:= Timer.Y;

END_FUNCTION_BLOCK

// Device/Application/Common_Functions/Pumphouse
FUNCTION_BLOCK Pumphouse
VAR_INPUT
END_VAR
VAR_OUTPUT
END_VAR
VAR
	//Fjernet logikblokk for pumpehus pga feilsøking.
	DrenPump	: SBE;
	ReturPump	: SBE;	
	Vippe_1		: MB;
	Vippe_2 	: MB; 
	Vippe_3		: MB;
END_VAR

Vippe_3(); // MB
Vippe_1(); // MB
Vippe_2(); // MB
DrenPump(); // SBE
Drenpump(); // SBE

END_FUNCTION_BLOCK

// Device/Application/Function blocks/Fault_Mapping
FUNCTION_BLOCK Fault_Mapping
VAR_INPUT
END_VAR
VAR_OUTPUT
END_VAR
VAR
END_VAR

END_FUNCTION_BLOCK

// Device/Application/Function blocks/fbBehandlaVatn
FUNCTION_BLOCK fbBehandlaVatn
VAR_INPUT
END_VAR
VAR_OUTPUT
END_VAR
VAR
END_VAR

END_FUNCTION_BLOCK

// Device/Application/Function blocks/fbFeilhandtering
FUNCTION_BLOCK fbFeilhandtering
VAR_INPUT
END_VAR
VAR_OUTPUT
END_VAR
VAR
END_VAR


// Collecting all faults to one fault output
// Here logic should be added what do when faults accur

END_FUNCTION_BLOCK

// Device/Application/Function blocks/fbPumphouse
FUNCTION_BLOCK fbPumphouse
VAR_INPUT
END_VAR
VAR_OUTPUT
END_VAR
VAR
END_VAR

END_FUNCTION_BLOCK

// Device/Application/Function blocks/fbPumpInterlock
FUNCTION_BLOCK fbPumpInterlock
VAR_INPUT
	X1					: BOOL;			// eXternal input1
	X2					: BOOL;			// eXternal input2
	XF					: BOOL;			// eXternal fault
END_VAR
VAR_OUTPUT
	Y1					: BOOL;			// Output
	Y2					: BOOL;			// Output
	YF					: BOOL;			// Output Fault
END_VAR

VAR
	Timer1				: fbTimer;		// Timer to hold the output
	Timer2				: fbTimer;		// Timer to hold the output
	sbX1				: BOOL;			// Static memory eXternal 
	sbX2				: BOOL;			// Static memory eXternal 
	siSwapCase		    : SINT;			// Static int Case
END_VAR

VAR_TEMP
	tbX1				: BOOL;			// temp eXternal input1
	tbX2				: BOOL;			// temp eXternal input2
	tbXF				: BOOL;			// eXternal fault			
	tbY1				: BOOL;			// temp output
	tbY2				: BOOL;			// temp output
END_VAR

VAR CONSTANT
	ciOutput1			: SINT := 1;		// constant case output 1
	ciOutput2			: SINT := 2;		// constant case output 2
	ciTimerT			: TIME := T#1s;		// Timedelay for output
END_VAR

// ***************************************************************************************
// Copyright: Peter Søreide Skaar, Roar Bøyum, Vegard Aven Ullebø [2024]
// All rights reserved.

// This code was developed as part of a Bachelor's thesis conducted for Renasys AS 
// and Sunnfjord Kommune. 

// Unauthorized reproduction, distribution, or modification of this code, in whole 
// or in part, is strictly prohibited without the express permission of the copyright 
// holder.
// ***************************************************************************************
// The code is used to interlock between reactors incase both are in pause sequence.
// Alternates the output if both inputs are high
// Else X1=Y1 and X2=Y2



// Populate temoraries
tbX1		:= X1;
tbX2		:= X2;
tbXF		:= XF;
tbY1		:= Y1;
tbY2		:= Y2;

Timer1();
Timer2();
Timer1.PTDH := ciTimerT;
Timer2.PTDH := ciTimerT;



// Handles if case is outside limits
IF (siSwapCase > ciOutput2) THEN
	siSwapCase := ciOutput1;
END_IF

// Handles if only one input is active
IF (tbX1 AND NOT tbX2) THEN
	tbY1 := TRUE;
ELSE
	tbY1 := FALSE;
END_IF

// Handles if only one input is active
IF (tbX2 AND NOT tbX1) THEN
	tbY2 := TRUE;
ELSE
	tbY2 := FALSE;
END_IF



// Handle Counter
// Counter increases by 1 each time Y2 goes high
IF tbX2 AND NOT sbX2 THEN
	siSwapCase := siSwapCase + 1;
END_IF

// Counter increases by 1 each time Y1 goes high
IF tbX1 AND NOT sbX1 THEN
	siSwapCase := siSwapCase + 1;
END_IF

// Retrigger posetive edge
sbX1						:= tbX1;	

// Retrigger posetive edge
sbX2						:= tbX2;	



//Check input, starts CASE
IF (tbX1 AND tbX2) THEN	

	CASE siSwapCase OF

		ciOutput1: // Statement section case 1 (Only Output Y1)	
			Timer1.X := TRUE;
			tbY2 := FALSE;
			tbY1 := TRUE;
	
// 			IF Timer1.Y THEN				
// 				tbY2 := FALSE;
// 				tbY1 := TRUE;
// 				Timer2.X 					:= FALSE;		
// 			END_IF
						

				
		ciOutput2: // Statement section case 2 (Only Output Y2)
			Timer2.X := TRUE;
			tbY1 := FALSE;
			tbY2 := TRUE;			
// 			IF Timer2.Y THEN				
// 
// 			Timer1.X 					:= FALSE;	
// 	
// 			END_IF

	END_CASE
END_IF





// Writing to outputs
Y1		:= tbY1;
Y2		:= tbY2;
YF		:= tbXF;

END_FUNCTION_BLOCK

// Device/Application/Functions/Volume_Rectangle
FUNCTION Volume_Rectangle : REAL
VAR_INPUT
	Height		: REAL;
	Widt		: REAL;
	Length		: REAL;
END_VAR
VAR_OUTPUT
	Volume		: REAL;
END_VAR
VAR
END_VAR

VAR CONSTANT

END_VAR

// ***************************************************************************************
// Copyright: Peter Søreide Skaar, Roar Bøyum, Vegard Aven Ullebø [2024]
// All rights reserved.

// This code was developed as part of a Bachelor's thesis conducted for Renasys AS 
// and Sunnfjord Kommune. 

// Unauthorized reproduction, distribution, or modification of this code, in whole 
// or in part, is strictly prohibited without the express permission of the copyright 
// holder.
// ***************************************************************************************


// This function calculates the volume of a rektangel
Volume := Height * Widt * Length;

END_FUNCTION

// Device/Application/Heile_R2/R2_Slam
FUNCTION_BLOCK R2_Slam
VAR_INPUT
	XE 			: BOOL;	
END_VAR
VAR_OUTPUT
END_VAR
VAR
	fbslamutak	: fbSlamUtak;
	PS01_VP01 	: SBV;
	PS00_VP01 	: SBV; //Sivebedventil 1
	PS00_VP02 	: SBV; //Sivebedventil 2
	PS00_VP03 	: SBV; //Sivebedventil 3
	PS00_VP04 	: SBV; //Sivebedventil 4
	
	Sim1		: fbValveSim;
	Sim2		: fbValveSim;
	Sim3		: fbValveSim;
	Sim4		: fbValveSim;
	Sim5		: fbValveSim;
	PS02_VP01: SBV;
END_VAR

